LIN {X 0,Y 361.866,Z 148.406,A -85,B 0,C 180,E1 -12924.654,E2 -12924.654} C_VEL
LIN {X 0,Y 361.829,Z 148.411,A -85,B 0,C 180,E1 -12928.369,E2 -12928.369} C_VEL
LIN {X 0,Y 361.892,Z 148.404,A -85,B 0,C 180,E1 -12930.954,E2 -12930.954} C_VEL
LIN {X 0,Y 361.9,Z 148.402,A -85,B 0,C 180,E1 -12934.708,E2 -12934.708} C_VEL
LIN {X 0,Y 361.851,Z 148.408,A -85,B 0,C 180,E1 -12938.344,E2 -12938.344} C_VEL
LIN {X 0,Y 361.91,Z 148.401,A -85,B 0,C 180,E1 -12942.084,E2 -12942.084} C_VEL
LIN {X 0,Y 361.95,Z 148.402,A -85,B 0,C 180,E1 -12945.379,E2 -12945.379} C_VEL
LIN {X 0,Y 361.958,Z 148.397,A -85,B 0,C 180,E1 -12948.804,E2 -12948.804} C_VEL
LIN {X 0,Y 362.066,Z 148.381,A -85,B 0,C 180,E1 -12952.191,E2 -12952.191} C_VEL
LIN {X 0,Y 362.076,Z 148.38,A -85,B 0,C 180,E1 -12954.43,E2 -12954.43} C_VEL
LIN {X 0,Y 362.251,Z 148.359,A -85,B 0,C 180,E1 -12957.776,E2 -12957.776} C_VEL
LIN {X 0,Y 362.252,Z 148.358,A -85,B 0,C 180,E1 -12962.224,E2 -12962.224} C_VEL
LIN {X 0,Y 362.111,Z 148.379,A -85,B 0,C 180,E1 -12966.687,E2 -12966.687} C_VEL
LIN {X 0,Y 361.988,Z 148.391,A -85,B 0,C 180,E1 -12970.063,E2 -12970.063} C_VEL
LIN {X 0,Y 361.987,Z 148.391,A -85,B 0,C 180,E1 -12973.899,E2 -12973.899} C_VEL
LIN {X 0,Y 361.917,Z 148.404,A -85,B 0,C 180,E1 -12976.935,E2 -12976.935} C_VEL
LIN {X 0,Y 361.876,Z 148.409,A -85,B 0,C 180,E1 -12980.462,E2 -12980.462} C_VEL
LIN {X 0,Y 361.883,Z 148.406,A -85,B 0,C 180,E1 -12984.113,E2 -12984.113} C_VEL
LIN {X 0,Y 361.889,Z 148.404,A -85,B 0,C 180,E1 -12987.781,E2 -12987.781} C_VEL
LIN {X 0,Y 361.837,Z 148.41,A -85,B 0,C 180,E1 -12991.286,E2 -12991.286} C_VEL
LIN {X 0,Y 361.845,Z 148.414,A -85,B 0,C 180,E1 -12994.281,E2 -12994.281} C_VEL
LIN {X 0,Y 361.854,Z 148.408,A -85,B 0,C 180,E1 -12997.224,E2 -12997.224} C_VEL
LIN {X 0,Y 361.827,Z 148.413,A -85,B 0,C 180,E1 -13000.756,E2 -13000.756} C_VEL
LIN {X 0,Y 361.81,Z 148.418,A -85,B 0,C 180,E1 -13004.37,E2 -13004.37} C_VEL
LIN {X 0,Y 361.83,Z 148.412,A -85,B 0,C 180,E1 -13007.569,E2 -13007.569} C_VEL
LIN {X 0,Y 361.864,Z 148.406,A -85,B 0,C 180,E1 -13010.975,E2 -13010.975} C_VEL
LIN {X 0,Y 361.87,Z 148.406,A -85,B 0,C 180,E1 -13014.657,E2 -13014.657} C_VEL
LIN {X 0,Y 361.834,Z 148.416,A -85,B 0,C 180,E1 -13018.372,E2 -13018.372} C_VEL
LIN {X 0,Y 361.897,Z 148.42,A -85,B 0,C 180,E1 -13020.133,E2 -13020.133} C_VEL
LIN {X 0,Y 364.194,Z 159.381,A -85,B 0,C 180,E1 -13022.801,E2 -13022.801} C_VEL
LIN {X 0,Y 365.334,Z 165.949,A -85,B 0,C 180,E1 -13024.346,E2 -13024.346} C_VEL
LIN {X 0,Y 364.928,Z 172.793,A -85,B 0,C 180,E1 -13025.844,E2 -13025.844} C_VEL
LIN {X 0,Y 363.854,Z 185.27,A -85,B 0,C 180,E1 -13028.536,E2 -13028.536} C_VEL
LIN {X 0,Y 368.797,Z 220.958,A -85,B 0,C 180,E1 -13029.526,E2 -13029.526} C_VEL
LIN {X 0,Y 367.709,Z 294.28,A -85,B 0,C 180,E1 -13030.971,E2 -13030.971} C_VEL
LIN {X 0,Y 367.075,Z 307.449,A -85,B 0,C 180,E1 -13031.441,E2 -13031.441} C_VEL
LIN {X 0,Y 366.307,Z 320.2,A -85,B 0,C 180,E1 -13032.124,E2 -13032.124} C_VEL
LIN {X 0,Y 365.392,Z 331.51,A -85,B 0,C 180,E1 -13032.944,E2 -13032.944} C_VEL
LIN {X 0,Y 364.323,Z 343.209,A -85,B 0,C 180,E1 -13034.046,E2 -13034.046} C_VEL
LIN {X 0,Y 363.402,Z 353.268,A -85,B 0,C 180,E1 -13035.234,E2 -13035.234} C_VEL
LIN {X 0,Y 362.556,Z 362.347,A -85,B 0,C 180,E1 -13036.55,E2 -13036.55} C_VEL
LIN {X 0,Y 361.857,Z 370.285,A -85,B 0,C 180,E1 -13037.95,E2 -13037.95} C_VEL
LIN {X 0,Y 361.155,Z 378.025,A -85,B 0,C 180,E1 -13039.631,E2 -13039.631} C_VEL
LIN {X 0,Y 360.675,Z 385.162,A -85,B 0,C 180,E1 -13041.598,E2 -13041.598} C_VEL
LIN {X 0,Y 360.482,Z 389.906,A -85,B 0,C 180,E1 -13043.283,E2 -13043.283} C_VEL
LIN {X 0,Y 360.379,Z 393.52,A -85,B 0,C 180,E1 -13044.966,E2 -13044.966} C_VEL
LIN {X 0,Y 360.356,Z 396.112,A -85,B 0,C 180,E1 -13046.647,E2 -13046.647} C_VEL
LIN {X 0,Y 360.396,Z 397.331,A -85,B 0,C 180,E1 -13047.766,E2 -13047.766} C_VEL
LIN {X 0,Y 360.461,Z 398.109,A -85,B 0,C 180,E1 -13048.884,E2 -13048.884} C_VEL
LIN {X 0,Y 360.481,Z 398.478,A -85,B 0,C 180,E1 -13050.001,E2 -13050.001} C_VEL
LIN {X 0,Y 360.456,Z 398.456,A -85,B 0,C 180,E1 -13051.118,E2 -13051.118} C_VEL
LIN {X 0,Y 360.353,Z 398.045,A -85,B 0,C 180,E1 -13052.236,E2 -13052.236} C_VEL
LIN {X 0,Y 360.325,Z 397.214,A -85,B 0,C 180,E1 -13053.355,E2 -13053.355} C_VEL
LIN {X 0,Y 360.36,Z 395.964,A -85,B 0,C 180,E1 -13054.475,E2 -13054.475} C_VEL
LIN {X 0,Y 360.378,Z 393.699,A -85,B 0,C 180,E1 -13055.962,E2 -13055.962} C_VEL
LIN {X 0,Y 360.611,Z 389.673,A -85,B 0,C 180,E1 -13057.842,E2 -13057.842} C_VEL
LIN {X 0,Y 360.997,Z 384.922,A -85,B 0,C 180,E1 -13059.526,E2 -13059.526} C_VEL
LIN {X 0,Y 361.76,Z 377.808,A -85,B 0,C 180,E1 -13061.487,E2 -13061.487} C_VEL
LIN {X 0,Y 362.786,Z 370.109,A -85,B 0,C 180,E1 -13063.158,E2 -13063.158} C_VEL
LIN {X 0,Y 363.776,Z 361.149,A -85,B 0,C 180,E1 -13064.722,E2 -13064.722} C_VEL
LIN {X 0,Y 364.888,Z 351.594,A -85,B 0,C 180,E1 -13066.074,E2 -13066.074} C_VEL
LIN {X 0,Y 366.215,Z 340.759,A -85,B 0,C 180,E1 -13067.306,E2 -13067.306} C_VEL
LIN {X 0,Y 367.436,Z 330.186,A -85,B 0,C 180,E1 -13068.253,E2 -13068.253} C_VEL
LIN {X 0,Y 368.413,Z 319.731,A -85,B 0,C 180,E1 -13068.996,E2 -13068.996} C_VEL
LIN {X 0,Y 369.47,Z 306.271,A -85,B 0,C 180,E1 -13069.698,E2 -13069.698} C_VEL
LIN {X 0,Y 370.177,Z 293.427,A -85,B 0,C 180,E1 -13070.14,E2 -13070.14} C_VEL
LIN {X 0,Y 371.381,Z 220.856,A -85,B 0,C 180,E1 -13071.578,E2 -13071.578} C_VEL
LIN {X 0,Y 366.879,Z 194.148,A -85,B 0,C 180,E1 -13072.44,E2 -13072.44} C_VEL
LIN {X 0,Y 365.076,Z 184.951,A -85,B 0,C 180,E1 -13072.766,E2 -13072.766} C_VEL
LIN {X 0,Y 366.595,Z 171.049,A -85,B 0,C 180,E1 -13075.824,E2 -13075.824} C_VEL
LIN {X 0,Y 365.256,Z 163.227,A -85,B 0,C 180,E1 -13077.736,E2 -13077.736} C_VEL
LIN {X 0,Y 362.77,Z 152.259,A -85,B 0,C 180,E1 -13080.551,E2 -13080.551} C_VEL
LIN {X 0,Y 361.907,Z 148.41,A -85,B 0,C 180,E1 -13081.623,E2 -13081.623} C_VEL
LIN {X 0,Y 361.87,Z 148.411,A -85,B 0,C 180,E1 -13085.637,E2 -13085.637} C_VEL
LIN {X 0,Y 361.866,Z 148.404,A -85,B 0,C 180,E1 -13089.026,E2 -13089.026} C_VEL
LIN {X 0,Y 361.838,Z 148.41,A -85,B 0,C 180,E1 -13092.829,E2 -13092.829} C_VEL
LIN {X 0,Y 361.82,Z 148.416,A -85,B 0,C 180,E1 -13095.947,E2 -13095.947} C_VEL
LIN {X 0,Y 361.814,Z 148.417,A -85,B 0,C 180,E1 -13099.249,E2 -13099.249} C_VEL
LIN {X 0,Y 361.864,Z 148.411,A -85,B 0,C 180,E1 -13102.982,E2 -13102.982} C_VEL
LIN {X 0,Y 361.859,Z 148.412,A -85,B 0,C 180,E1 -13106.631,E2 -13106.631} C_VEL
LIN {X 0,Y 361.857,Z 148.409,A -85,B 0,C 180,E1 -13109.67,E2 -13109.67} C_VEL
LIN {X 0,Y 361.864,Z 148.407,A -85,B 0,C 180,E1 -13113.468,E2 -13113.468} C_VEL
LIN {X 0,Y 361.865,Z 148.409,A -85,B 0,C 180,E1 -13117.143,E2 -13117.143} C_VEL
LIN {X 0,Y 361.855,Z 148.403,A -85,B 0,C 180,E1 -13120.721,E2 -13120.721} C_VEL
LIN {X 0,Y 361.89,Z 148.406,A -85,B 0,C 180,E1 -13124.224,E2 -13124.224} C_VEL
LIN {X 0,Y 361.999,Z 148.386,A -85,B 0,C 180,E1 -13126.528,E2 -13126.528} C_VEL
LIN {X 0,Y 361.994,Z 148.393,A -85,B 0,C 180,E1 -13129.937,E2 -13129.937} C_VEL
LIN {X 0,Y 362.118,Z 148.374,A -85,B 0,C 180,E1 -13133.313,E2 -13133.313} C_VEL
LIN {X 0,Y 362.257,Z 148.351,A -85,B 0,C 180,E1 -13137.776,E2 -13137.776} C_VEL
LIN {X 0,Y 362.173,Z 148.369,A -85,B 0,C 180,E1 -13141.112,E2 -13141.112} C_VEL
LIN {X 0,Y 362.258,Z 148.351,A -85,B 0,C 180,E1 -13142.224,E2 -13142.224} C_VEL
LIN {X 0,Y 362.122,Z 148.374,A -85,B 0,C 180,E1 -13146.687,E2 -13146.687} C_VEL
LIN {X 0,Y 362.001,Z 148.391,A -85,B 0,C 180,E1 -13150.063,E2 -13150.063} C_VEL
LIN {X 0,Y 362,Z 148.382,A -85,B 0,C 180,E1 -13153.899,E2 -13153.899} C_VEL
LIN {X 0,Y 361.929,Z 148.401,A -85,B 0,C 180,E1 -13156.934,E2 -13156.934} C_VEL
LIN {X 0,Y 361.885,Z 148.4,A -85,B 0,C 180,E1 -13160.461,E2 -13160.461} C_VEL
LIN {X 0,Y 361.896,Z 148.397,A -85,B 0,C 180,E1 -13164.113,E2 -13164.113} C_VEL
LIN {X 0,Y 361.863,Z 148.405,A -85,B 0,C 180,E1 -13167.783,E2 -13167.783} C_VEL
LIN {X 0,Y 361.849,Z 148.41,A -85,B 0,C 180,E1 -13171.285,E2 -13171.285} C_VEL
LIN {X 0,Y 361.857,Z 148.409,A -85,B 0,C 180,E1 -13174.28,E2 -13174.28} C_VEL
LIN {X 0,Y 361.865,Z 148.408,A -85,B 0,C 180,E1 -13177.223,E2 -13177.223} C_VEL
LIN {X 0,Y 361.837,Z 148.396,A -85,B 0,C 180,E1 -13180.755,E2 -13180.755} C_VEL
LIN {X 0,Y 361.821,Z 148.416,A -85,B 0,C 180,E1 -13184.368,E2 -13184.368} C_VEL
LIN {X 0,Y 361.836,Z 148.411,A -85,B 0,C 180,E1 -13187.569,E2 -13187.569} C_VEL
LIN {X 0,Y 361.869,Z 148.408,A -85,B 0,C 180,E1 -13190.974,E2 -13190.974} C_VEL
LIN {X 0,Y 361.878,Z 148.408,A -85,B 0,C 180,E1 -13194.655,E2 -13194.655} C_VEL
LIN {X 0,Y 361.842,Z 148.409,A -85,B 0,C 180,E1 -13198.37,E2 -13198.37} C_VEL
LIN {X 0,Y 361.894,Z 148.509,A -85,B 0,C 180,E1 -13200.234,E2 -13200.234} C_VEL
LIN {X 0,Y 363.473,Z 155.472,A -85,B 0,C 180,E1 -13202.171,E2 -13202.171} C_VEL
LIN {X 0,Y 370.386,Z 172.492,A -85,B 0,C 180,E1 -13203.028,E2 -13203.028} C_VEL
LIN {X 0,Y 372.236,Z 181.018,A -85,B 0,C 180,E1 -13203.333,E2 -13203.333} C_VEL
LIN {X 0,Y 370.673,Z 262.367,A -85,B 0,C 180,E1 -13204.935,E2 -13204.935} C_VEL
LIN {X 0,Y 370.018,Z 275.946,A -85,B 0,C 180,E1 -13205.424,E2 -13205.424} C_VEL
LIN {X 0,Y 369.16,Z 288.919,A -85,B 0,C 180,E1 -13206.13,E2 -13206.13} C_VEL
LIN {X 0,Y 368.348,Z 300.168,A -85,B 0,C 180,E1 -13206.974,E2 -13206.974} C_VEL
LIN {X 0,Y 367.174,Z 311.746,A -85,B 0,C 180,E1 -13208.083,E2 -13208.083} C_VEL
LIN {X 0,Y 366.036,Z 321.067,A -85,B 0,C 180,E1 -13209.193,E2 -13209.193} C_VEL
LIN {X 0,Y 364.942,Z 331.045,A -85,B 0,C 180,E1 -13210.672,E2 -13210.672} C_VEL
LIN {X 0,Y 363.824,Z 339.748,A -85,B 0,C 180,E1 -13212.287,E2 -13212.287} C_VEL
LIN {X 0,Y 362.789,Z 347.08,A -85,B 0,C 180,E1 -13213.974,E2 -13213.974} C_VEL
LIN {X 0,Y 361.91,Z 353.714,A -85,B 0,C 180,E1 -13215.931,E2 -13215.931} C_VEL
LIN {X 0,Y 361.358,Z 358.166,A -85,B 0,C 180,E1 -13217.646,E2 -13217.646} C_VEL
LIN {X 0,Y 361.008,Z 360.482,A -85,B 0,C 180,E1 -13218.773,E2 -13218.773} C_VEL
LIN {X 0,Y 360.793,Z 362.366,A -85,B 0,C 180,E1 -13219.902,E2 -13219.902} C_VEL
LIN {X 0,Y 360.655,Z 363.801,A -85,B 0,C 180,E1 -13221.03,E2 -13221.03} C_VEL
LIN {X 0,Y 360.563,Z 365.424,A -85,B 0,C 180,E1 -13223.283,E2 -13223.283} C_VEL
LIN {X 0,Y 360.503,Z 365.665,A -85,B 0,C 180,E1 -13224.405,E2 -13224.405} C_VEL
LIN {X 0,Y 360.478,Z 365.493,A -85,B 0,C 180,E1 -13225.526,E2 -13225.526} C_VEL
LIN {X 0,Y 360.495,Z 363.954,A -85,B 0,C 180,E1 -13227.764,E2 -13227.764} C_VEL
LIN {X 0,Y 360.56,Z 362.608,A -85,B 0,C 180,E1 -13228.882,E2 -13228.882} C_VEL
LIN {X 0,Y 360.722,Z 359.766,A -85,B 0,C 180,E1 -13230.557,E2 -13230.557} C_VEL
LIN {X 0,Y 360.976,Z 355.915,A -85,B 0,C 180,E1 -13232.231,E2 -13232.231} C_VEL
LIN {X 0,Y 361.501,Z 350.939,A -85,B 0,C 180,E1 -13233.901,E2 -13233.901} C_VEL
LIN {X 0,Y 362.073,Z 344.7,A -85,B 0,C 180,E1 -13235.568,E2 -13235.568} C_VEL
LIN {X 0,Y 362.934,Z 336.878,A -85,B 0,C 180,E1 -13237.23,E2 -13237.23} C_VEL
LIN {X 0,Y 363.748,Z 328.918,A -85,B 0,C 180,E1 -13238.611,E2 -13238.611} C_VEL
LIN {X 0,Y 364.686,Z 319.213,A -85,B 0,C 180,E1 -13239.987,E2 -13239.987} C_VEL
LIN {X 0,Y 365.617,Z 308.385,A -85,B 0,C 180,E1 -13241.222,E2 -13241.222} C_VEL
LIN {X 0,Y 366.453,Z 297.773,A -85,B 0,C 180,E1 -13242.178,E2 -13242.178} C_VEL
LIN {X 0,Y 367.184,Z 285.026,A -85,B 0,C 180,E1 -13243.066,E2 -13243.066} C_VEL
LIN {X 0,Y 367.793,Z 272.056,A -85,B 0,C 180,E1 -13243.712,E2 -13243.712} C_VEL
LIN {X 0,Y 368.128,Z 259.143,A -85,B 0,C 180,E1 -13244.122,E2 -13244.122} C_VEL
LIN {X 0,Y 368.76,Z 224.019,A -85,B 0,C 180,E1 -13244.807,E2 -13244.807} C_VEL
LIN {X 0,Y 368.211,Z 218.205,A -85,B 0,C 180,E1 -13244.952,E2 -13244.952} C_VEL
LIN {X 0,Y 363.043,Z 199.491,A -85,B 0,C 180,E1 -13245.605,E2 -13245.605} C_VEL
LIN {X 0,Y 362.507,Z 193.676,A -85,B 0,C 180,E1 -13245.754,E2 -13245.754} C_VEL
LIN {X 0,Y 362.662,Z 178.93,A -85,B 0,C 180,E1 -13246.048,E2 -13246.048} C_VEL
LIN {X 0,Y 359.731,Z 165.344,A -85,B 0,C 180,E1 -13246.495,E2 -13246.495} C_VEL
LIN {X 0,Y 356.068,Z 155.147,A -85,B 0,C 180,E1 -13246.938,E2 -13246.938} C_VEL
LIN {X 0,Y 354.923,Z 149.276,A -85,B 0,C 180,E1 -13248.582,E2 -13248.582} C_VEL
LIN {X 0,Y 354.815,Z 149.288,A -85,B 0,C 180,E1 -13252.106,E2 -13252.106} C_VEL
LIN {X 0,Y 354.897,Z 149.276,A -85,B 0,C 180,E1 -13255.826,E2 -13255.826} C_VEL
LIN {X 0,Y 354.852,Z 149.281,A -85,B 0,C 180,E1 -13259.677,E2 -13259.677} C_VEL
LIN {X 0,Y 354.803,Z 149.288,A -85,B 0,C 180,E1 -13263.701,E2 -13263.701} C_VEL
LIN {X 0,Y 354.795,Z 149.289,A -85,B 0,C 180,E1 -13266.458,E2 -13266.458} C_VEL
LIN {X 0,Y 354.82,Z 149.285,A -85,B 0,C 180,E1 -13269.422,E2 -13269.422} C_VEL
LIN {X 0,Y 354.783,Z 149.288,A -85,B 0,C 180,E1 -13272.866,E2 -13272.866} C_VEL
LIN {X 0,Y 354.761,Z 149.295,A -85,B 0,C 180,E1 -13276.102,E2 -13276.102} C_VEL
LIN {X 0,Y 354.781,Z 149.289,A -85,B 0,C 180,E1 -13279.178,E2 -13279.178} C_VEL
LIN {X 0,Y 354.799,Z 149.287,A -85,B 0,C 180,E1 -13282.402,E2 -13282.402} C_VEL
LIN {X 0,Y 354.804,Z 149.286,A -85,B 0,C 180,E1 -13284.94,E2 -13284.94} C_VEL
LIN {X 0,Y 354.785,Z 149.288,A -85,B 0,C 180,E1 -13288.404,E2 -13288.404} C_VEL
LIN {X 0,Y 354.831,Z 149.288,A -85,B 0,C 180,E1 -13291.617,E2 -13291.617} C_VEL
LIN {X 0,Y 354.865,Z 149.279,A -85,B 0,C 180,E1 -13294.17,E2 -13294.17} C_VEL
LIN {X 0,Y 354.805,Z 149.287,A -85,B 0,C 180,E1 -13297.892,E2 -13297.892} C_VEL
LIN {X 0,Y 354.88,Z 149.278,A -85,B 0,C 180,E1 -13301.907,E2 -13301.907} C_VEL
LIN {X 0,Y 354.932,Z 149.27,A -85,B 0,C 180,E1 -13305.981,E2 -13305.981} C_VEL
LIN {X 0,Y 354.944,Z 149.27,A -85,B 0,C 180,E1 -13309.735,E2 -13309.735} C_VEL
LIN {X 0,Y 355.073,Z 149.258,A -85,B 0,C 180,E1 -13313.179,E2 -13313.179} C_VEL
LIN {X 0,Y 355.213,Z 149.235,A -85,B 0,C 180,E1 -13317.732,E2 -13317.732} C_VEL
LIN {X 0,Y 355.133,Z 149.25,A -85,B 0,C 180,E1 -13321.134,E2 -13321.134} C_VEL
LIN {X 0,Y 355.214,Z 149.235,A -85,B 0,C 180,E1 -13322.268,E2 -13322.268} C_VEL
LIN {X 0,Y 355.076,Z 149.257,A -85,B 0,C 180,E1 -13326.82,E2 -13326.82} C_VEL
LIN {X 0,Y 354.944,Z 149.269,A -85,B 0,C 180,E1 -13330.265,E2 -13330.265} C_VEL
LIN {X 0,Y 354.932,Z 149.27,A -85,B 0,C 180,E1 -13334.019,E2 -13334.019} C_VEL
LIN {X 0,Y 354.879,Z 149.277,A -85,B 0,C 180,E1 -13338.093,E2 -13338.093} C_VEL
LIN {X 0,Y 354.805,Z 149.287,A -85,B 0,C 180,E1 -13342.108,E2 -13342.108} C_VEL
LIN {X 0,Y 354.865,Z 149.278,A -85,B 0,C 180,E1 -13345.83,E2 -13345.83} C_VEL
LIN {X 0,Y 354.845,Z 149.281,A -85,B 0,C 180,E1 -13349.679,E2 -13349.679} C_VEL
LIN {X 0,Y 354.798,Z 149.287,A -85,B 0,C 180,E1 -13353.703,E2 -13353.703} C_VEL
LIN {X 0,Y 354.789,Z 149.293,A -85,B 0,C 180,E1 -13356.461,E2 -13356.461} C_VEL
LIN {X 0,Y 354.816,Z 149.284,A -85,B 0,C 180,E1 -13359.425,E2 -13359.425} C_VEL
LIN {X 0,Y 354.781,Z 149.289,A -85,B 0,C 180,E1 -13362.868,E2 -13362.868} C_VEL
LIN {X 0,Y 354.761,Z 149.297,A -85,B 0,C 180,E1 -13366.105,E2 -13366.105} C_VEL
LIN {X 0,Y 354.782,Z 149.288,A -85,B 0,C 180,E1 -13369.18,E2 -13369.18} C_VEL
LIN {X 0,Y 354.802,Z 149.289,A -85,B 0,C 180,E1 -13372.404,E2 -13372.404} C_VEL
LIN {X 0,Y 354.807,Z 149.285,A -85,B 0,C 180,E1 -13374.942,E2 -13374.942} C_VEL
LIN {X 0,Y 354.79,Z 149.294,A -85,B 0,C 180,E1 -13378.406,E2 -13378.406} C_VEL
LIN {X 0,Y 354.854,Z 149.345,A -85,B 0,C 180,E1 -13379.832,E2 -13379.832} C_VEL
LIN {X 0,Y 357.322,Z 161.045,A -85,B 0,C 180,E1 -13382.742,E2 -13382.742} C_VEL
LIN {X 0,Y 358.436,Z 168.19,A -85,B 0,C 180,E1 -13384.447,E2 -13384.447} C_VEL
LIN {X 0,Y 357.165,Z 182.663,A -85,B 0,C 180,E1 -13387.643,E2 -13387.643} C_VEL
LIN {X 0,Y 356.935,Z 184.932,A -85,B 0,C 180,E1 -13388.139,E2 -13388.139} C_VEL
LIN {X 0,Y 361.814,Z 219.463,A -85,B 0,C 180,E1 -13389.13,E2 -13389.13} C_VEL
LIN {X 0,Y 362.034,Z 226.1,A -85,B 0,C 180,E1 -13389.278,E2 -13389.278} C_VEL
LIN {X 0,Y 360.934,Z 293.87,A -85,B 0,C 180,E1 -13390.637,E2 -13390.637} C_VEL
LIN {X 0,Y 360.284,Z 307.058,A -85,B 0,C 180,E1 -13391.115,E2 -13391.115} C_VEL
LIN {X 0,Y 359.516,Z 319.257,A -85,B 0,C 180,E1 -13391.775,E2 -13391.775} C_VEL
LIN {X 0,Y 358.596,Z 330.743,A -85,B 0,C 180,E1 -13392.611,E2 -13392.611} C_VEL
LIN {X 0,Y 357.472,Z 342.534,A -85,B 0,C 180,E1 -13393.732,E2 -13393.732} C_VEL
LIN {X 0,Y 356.386,Z 353.719,A -85,B 0,C 180,E1 -13395.081,E2 -13395.081} C_VEL
LIN {X 0,Y 355.631,Z 361.782,A -85,B 0,C 180,E1 -13396.283,E2 -13396.283} C_VEL
LIN {X 0,Y 354.866,Z 369.76,A -85,B 0,C 180,E1 -13397.709,E2 -13397.709} C_VEL
LIN {X 0,Y 354.123,Z 377.548,A -85,B 0,C 180,E1 -13399.423,E2 -13399.423} C_VEL
LIN {X 0,Y 353.619,Z 384.715,A -85,B 0,C 180,E1 -13401.429,E2 -13401.429} C_VEL
LIN {X 0,Y 353.392,Z 389.484,A -85,B 0,C 180,E1 -13403.148,E2 -13403.148} C_VEL
LIN {X 0,Y 353.282,Z 393.124,A -85,B 0,C 180,E1 -13404.865,E2 -13404.865} C_VEL
LIN {X 0,Y 353.275,Z 395.74,A -85,B 0,C 180,E1 -13406.58,E2 -13406.58} C_VEL
LIN {X 0,Y 353.297,Z 396.971,A -85,B 0,C 180,E1 -13407.721,E2 -13407.721} C_VEL
LIN {X 0,Y 353.364,Z 397.769,A -85,B 0,C 180,E1 -13408.861,E2 -13408.861} C_VEL
LIN {X 0,Y 353.4,Z 398.149,A -85,B 0,C 180,E1 -13410.001,E2 -13410.001} C_VEL
LIN {X 0,Y 353.357,Z 398.137,A -85,B 0,C 180,E1 -13411.141,E2 -13411.141} C_VEL
LIN {X 0,Y 353.255,Z 397.737,A -85,B 0,C 180,E1 -13412.281,E2 -13412.281} C_VEL
LIN {X 0,Y 353.244,Z 396.927,A -85,B 0,C 180,E1 -13413.423,E2 -13413.423} C_VEL
LIN {X 0,Y 353.27,Z 395.688,A -85,B 0,C 180,E1 -13414.565,E2 -13414.565} C_VEL
LIN {X 0,Y 353.272,Z 393.744,A -85,B 0,C 180,E1 -13415.899,E2 -13415.899} C_VEL
LIN {X 0,Y 353.548,Z 389.443,A -85,B 0,C 180,E1 -13418,E2 -13418} C_VEL
LIN {X 0,Y 353.97,Z 384.717,A -85,B 0,C 180,E1 -13419.717,E2 -13419.717} C_VEL
LIN {X 0,Y 354.775,Z 377.633,A -85,B 0,C 180,E1 -13421.716,E2 -13421.716} C_VEL
LIN {X 0,Y 355.85,Z 369.978,A -85,B 0,C 180,E1 -13423.419,E2 -13423.419} C_VEL
LIN {X 0,Y 356.952,Z 360.632,A -85,B 0,C 180,E1 -13425.081,E2 -13425.081} C_VEL
LIN {X 0,Y 358.213,Z 350.491,A -85,B 0,C 180,E1 -13426.529,E2 -13426.529} C_VEL
LIN {X 0,Y 359.622,Z 339.415,A -85,B 0,C 180,E1 -13427.78,E2 -13427.78} C_VEL
LIN {X 0,Y 360.884,Z 328.579,A -85,B 0,C 180,E1 -13428.744,E2 -13428.744} C_VEL
LIN {X 0,Y 362.059,Z 316.639,A -85,B 0,C 180,E1 -13429.564,E2 -13429.564} C_VEL
LIN {X 0,Y 363.022,Z 303.678,A -85,B 0,C 180,E1 -13430.21,E2 -13430.21} C_VEL
LIN {X 0,Y 363.649,Z 290.822,A -85,B 0,C 180,E1 -13430.617,E2 -13430.617} C_VEL
LIN {X 0,Y 364.924,Z 222.57,A -85,B 0,C 180,E1 -13431.978,E2 -13431.978} C_VEL
LIN {X 0,Y 360.899,Z 197.766,A -85,B 0,C 180,E1 -13432.788,E2 -13432.788} C_VEL
LIN {X 0,Y 358.307,Z 184.595,A -85,B 0,C 180,E1 -13433.27,E2 -13433.27} C_VEL
LIN {X 0,Y 359.724,Z 172.373,A -85,B 0,C 180,E1 -13436.011,E2 -13436.011} C_VEL
LIN {X 0,Y 357.952,Z 162.741,A -85,B 0,C 180,E1 -13438.433,E2 -13438.433} C_VEL
LIN {X 0,Y 354.854,Z 149.29,A -85,B 0,C 180,E1 -13442.02,E2 -13442.02} C_VEL
LIN {X 0,Y 354.824,Z 149.29,A -85,B 0,C 180,E1 -13445.7,E2 -13445.7} C_VEL
LIN {X 0,Y 354.827,Z 149.281,A -85,B 0,C 180,E1 -13449.424,E2 -13449.424} C_VEL
LIN {X 0,Y 354.79,Z 149.288,A -85,B 0,C 180,E1 -13452.867,E2 -13452.867} C_VEL
LIN {X 0,Y 354.768,Z 149.293,A -85,B 0,C 180,E1 -13456.104,E2 -13456.104} C_VEL
LIN {X 0,Y 354.767,Z 149.295,A -85,B 0,C 180,E1 -13459.176,E2 -13459.176} C_VEL
LIN {X 0,Y 354.801,Z 149.289,A -85,B 0,C 180,E1 -13462.405,E2 -13462.405} C_VEL
LIN {X 0,Y 354.81,Z 149.29,A -85,B 0,C 180,E1 -13464.941,E2 -13464.941} C_VEL
LIN {X 0,Y 354.795,Z 149.29,A -85,B 0,C 180,E1 -13468.405,E2 -13468.405} C_VEL
LIN {X 0,Y 354.801,Z 149.287,A -85,B 0,C 180,E1 -13471.615,E2 -13471.615} C_VEL
LIN {X 0,Y 354.836,Z 149.283,A -85,B 0,C 180,E1 -13475.657,E2 -13475.657} C_VEL
LIN {X 0,Y 354.822,Z 149.281,A -85,B 0,C 180,E1 -13479.113,E2 -13479.113} C_VEL
LIN {X 0,Y 354.852,Z 149.284,A -85,B 0,C 180,E1 -13482.718,E2 -13482.718} C_VEL
LIN {X 0,Y 354.94,Z 149.263,A -85,B 0,C 180,E1 -13486.255,E2 -13486.255} C_VEL
LIN {X 0,Y 354.95,Z 149.27,A -85,B 0,C 180,E1 -13489.735,E2 -13489.735} C_VEL
LIN {X 0,Y 355.085,Z 149.25,A -85,B 0,C 180,E1 -13493.18,E2 -13493.18} C_VEL
LIN {X 0,Y 355.218,Z 149.227,A -85,B 0,C 180,E1 -13497.732,E2 -13497.732} C_VEL
LIN {X 0,Y 355.145,Z 149.244,A -85,B 0,C 180,E1 -13501.134,E2 -13501.134} C_VEL
LIN {X 0,Y 355.22,Z 149.227,A -85,B 0,C 180,E1 -13502.268,E2 -13502.268} C_VEL
LIN {X 0,Y 355.088,Z 149.251,A -85,B 0,C 180,E1 -13506.82,E2 -13506.82} C_VEL
LIN {X 0,Y 354.957,Z 149.267,A -85,B 0,C 180,E1 -13510.265,E2 -13510.265} C_VEL
LIN {X 0,Y 354.945,Z 149.26,A -85,B 0,C 180,E1 -13514.019,E2 -13514.019} C_VEL
LIN {X 0,Y 354.892,Z 149.274,A -85,B 0,C 180,E1 -13518.092,E2 -13518.092} C_VEL
LIN {X 0,Y 354.817,Z 149.285,A -85,B 0,C 180,E1 -13522.107,E2 -13522.107} C_VEL
LIN {X 0,Y 354.828,Z 149.284,A -85,B 0,C 180,E1 -13525.833,E2 -13525.833} C_VEL
LIN {X 0,Y 354.81,Z 149.285,A -85,B 0,C 180,E1 -13529.683,E2 -13529.683} C_VEL
LIN {X 0,Y 354.817,Z 149.284,A -85,B 0,C 180,E1 -13533.684,E2 -13533.684} C_VEL
LIN {X 0,Y 354.8,Z 149.286,A -85,B 0,C 180,E1 -13536.46,E2 -13536.46} C_VEL
LIN {X 0,Y 354.827,Z 149.28,A -85,B 0,C 180,E1 -13539.424,E2 -13539.424} C_VEL
LIN {X 0,Y 354.791,Z 149.287,A -85,B 0,C 180,E1 -13542.867,E2 -13542.867} C_VEL
LIN {X 0,Y 354.77,Z 149.294,A -85,B 0,C 180,E1 -13546.103,E2 -13546.103} C_VEL
LIN {X 0,Y 354.787,Z 149.29,A -85,B 0,C 180,E1 -13549.178,E2 -13549.178} C_VEL
LIN {X 0,Y 354.81,Z 149.289,A -85,B 0,C 180,E1 -13552.403,E2 -13552.403} C_VEL
LIN {X 0,Y 354.816,Z 149.288,A -85,B 0,C 180,E1 -13554.941,E2 -13554.941} C_VEL
LIN {X 0,Y 354.797,Z 149.287,A -85,B 0,C 180,E1 -13558.405,E2 -13558.405} C_VEL
LIN {X 0,Y 354.872,Z 149.464,A -85,B 0,C 180,E1 -13559.831,E2 -13559.831} C_VEL
LIN {X 0,Y 356.321,Z 155.683,A -85,B 0,C 180,E1 -13561.634,E2 -13561.634} C_VEL
LIN {X 0,Y 364.068,Z 174.56,A -85,B 0,C 180,E1 -13562.622,E2 -13562.622} C_VEL
LIN {X 0,Y 365.745,Z 181.421,A -85,B 0,C 180,E1 -13562.888,E2 -13562.888} C_VEL
LIN {X 0,Y 364.092,Z 263.039,A -85,B 0,C 180,E1 -13564.526,E2 -13564.526} C_VEL
LIN {X 0,Y 363.43,Z 276.633,A -85,B 0,C 180,E1 -13565.031,E2 -13565.031} C_VEL
LIN {X 0,Y 362.618,Z 288.293,A -85,B 0,C 180,E1 -13565.671,E2 -13565.671} C_VEL
LIN {X 0,Y 361.77,Z 299.814,A -85,B 0,C 180,E1 -13566.531,E2 -13566.531} C_VEL
LIN {X 0,Y 360.546,Z 311.518,A -85,B 0,C 180,E1 -13567.659,E2 -13567.659} C_VEL
LIN {X 0,Y 359.359,Z 320.934,A -85,B 0,C 180,E1 -13568.788,E2 -13568.788} C_VEL
LIN {X 0,Y 358.199,Z 330.74,A -85,B 0,C 180,E1 -13570.247,E2 -13570.247} C_VEL
LIN {X 0,Y 357.006,Z 339.784,A -85,B 0,C 180,E1 -13571.937,E2 -13571.937} C_VEL
LIN {X 0,Y 355.913,Z 347.167,A -85,B 0,C 180,E1 -13573.656,E2 -13573.656} C_VEL
LIN {X 0,Y 355.163,Z 352.164,A -85,B 0,C 180,E1 -13575.092,E2 -13575.092} C_VEL
LIN {X 0,Y 354.502,Z 356.994,A -85,B 0,C 180,E1 -13576.821,E2 -13576.821} C_VEL
LIN {X 0,Y 354.008,Z 360.693,A -85,B 0,C 180,E1 -13578.548,E2 -13578.548} C_VEL
LIN {X 0,Y 353.739,Z 362.596,A -85,B 0,C 180,E1 -13579.699,E2 -13579.699} C_VEL
LIN {X 0,Y 353.587,Z 364.065,A -85,B 0,C 180,E1 -13580.85,E2 -13580.85} C_VEL
LIN {X 0,Y 353.49,Z 365.722,A -85,B 0,C 180,E1 -13583.148,E2 -13583.148} C_VEL
LIN {X 0,Y 353.427,Z 365.98,A -85,B 0,C 180,E1 -13584.293,E2 -13584.293} C_VEL
LIN {X 0,Y 353.409,Z 365.841,A -85,B 0,C 180,E1 -13585.437,E2 -13585.437} C_VEL
LIN {X 0,Y 353.397,Z 364.338,A -85,B 0,C 180,E1 -13587.72,E2 -13587.72} C_VEL
LIN {X 0,Y 353.493,Z 363.007,A -85,B 0,C 180,E1 -13588.86,E2 -13588.86} C_VEL
LIN {X 0,Y 353.639,Z 360.203,A -85,B 0,C 180,E1 -13590.568,E2 -13590.568} C_VEL
LIN {X 0,Y 353.908,Z 356.39,A -85,B 0,C 180,E1 -13592.275,E2 -13592.275} C_VEL
LIN {X 0,Y 354.432,Z 351.455,A -85,B 0,C 180,E1 -13593.978,E2 -13593.978} C_VEL
LIN {X 0,Y 355.05,Z 345.266,A -85,B 0,C 180,E1 -13595.679,E2 -13595.679} C_VEL
LIN {X 0,Y 355.937,Z 337.515,A -85,B 0,C 180,E1 -13597.373,E2 -13597.373} C_VEL
LIN {X 0,Y 356.772,Z 329.617,A -85,B 0,C 180,E1 -13598.78,E2 -13598.78} C_VEL
LIN {X 0,Y 357.819,Z 318.987,A -85,B 0,C 180,E1 -13600.316,E2 -13600.316} C_VEL
LIN {X 0,Y 358.77,Z 308.181,A -85,B 0,C 180,E1 -13601.553,E2 -13601.553} C_VEL
LIN {X 0,Y 359.705,Z 297.088,A -85,B 0,C 180,E1 -13602.553,E2 -13602.553} C_VEL
LIN {X 0,Y 360.38,Z 285.183,A -85,B 0,C 180,E1 -13603.389,E2 -13603.389} C_VEL
LIN {X 0,Y 360.993,Z 272.982,A -85,B 0,C 180,E1 -13604.012,E2 -13604.012} C_VEL
LIN {X 0,Y 361.347,Z 260.511,A -85,B 0,C 180,E1 -13604.429,E2 -13604.429} C_VEL
LIN {X 0,Y 362.507,Z 193.676,A -85,B 0,C 180,E1 -13605.754,E2 -13605.754} C_VEL
LIN {X 0,Y 361.897,Z 187.877,A -85,B 0,C 180,E1 -13605.906,E2 -13605.906} C_VEL
LIN {X 0,Y 360.221,Z 182.318,A -85,B 0,C 180,E1 -13606.115,E2 -13606.115} C_VEL
LIN {X 0,Y 352.169,Z 164.496,A -85,B 0,C 180,E1 -13606.957,E2 -13606.957} C_VEL
LIN {X 0,Y 348.908,Z 155.398,A -85,B 0,C 180,E1 -13607.385,E2 -13607.385} C_VEL
LIN {X 0,Y 347.874,Z 150.152,A -85,B 0,C 180,E1 -13608.858,E2 -13608.858} C_VEL
LIN {X 0,Y 347.762,Z 150.167,A -85,B 0,C 180,E1 -13612.579,E2 -13612.579} C_VEL
LIN {X 0,Y 347.81,Z 150.157,A -85,B 0,C 180,E1 -13615.107,E2 -13615.107} C_VEL
LIN {X 0,Y 347.809,Z 150.159,A -85,B 0,C 180,E1 -13617.692,E2 -13617.692} C_VEL
LIN {X 0,Y 347.762,Z 150.167,A -85,B 0,C 180,E1 -13620.345,E2 -13620.345} C_VEL
LIN {X 0,Y 347.741,Z 150.168,A -85,B 0,C 180,E1 -13624.462,E2 -13624.462} C_VEL
LIN {X 0,Y 347.77,Z 150.168,A -85,B 0,C 180,E1 -13627.987,E2 -13627.987} C_VEL
LIN {X 0,Y 347.746,Z 150.17,A -85,B 0,C 180,E1 -13631.829,E2 -13631.829} C_VEL
LIN {X 0,Y 347.7,Z 150.171,A -85,B 0,C 180,E1 -13635.025,E2 -13635.025} C_VEL
LIN {X 0,Y 347.744,Z 150.166,A -85,B 0,C 180,E1 -13638.396,E2 -13638.396} C_VEL
LIN {X 0,Y 347.766,Z 150.166,A -85,B 0,C 180,E1 -13642.01,E2 -13642.01} C_VEL
LIN {X 0,Y 347.736,Z 150.171,A -85,B 0,C 180,E1 -13645.535,E2 -13645.535} C_VEL
LIN {X 0,Y 347.755,Z 150.17,A -85,B 0,C 180,E1 -13649.652,E2 -13649.652} C_VEL
LIN {X 0,Y 347.814,Z 150.156,A -85,B 0,C 180,E1 -13652.753,E2 -13652.753} C_VEL
LIN {X 0,Y 347.774,Z 150.162,A -85,B 0,C 180,E1 -13656.161,E2 -13656.161} C_VEL
LIN {X 0,Y 347.789,Z 150.161,A -85,B 0,C 180,E1 -13659.908,E2 -13659.908} C_VEL
LIN {X 0,Y 347.82,Z 150.159,A -85,B 0,C 180,E1 -13663.568,E2 -13663.568} C_VEL
LIN {X 0,Y 347.878,Z 150.153,A -85,B 0,C 180,E1 -13667.16,E2 -13667.16} C_VEL
LIN {X 0,Y 347.924,Z 150.144,A -85,B 0,C 180,E1 -13670.7,E2 -13670.7} C_VEL
LIN {X 0,Y 348.024,Z 150.128,A -85,B 0,C 180,E1 -13674.205,E2 -13674.205} C_VEL
LIN {X 0,Y 348.175,Z 150.112,A -85,B 0,C 180,E1 -13677.686,E2 -13677.686} C_VEL
LIN {X 0,Y 348.104,Z 150.125,A -85,B 0,C 180,E1 -13681.157,E2 -13681.157} C_VEL
LIN {X 0,Y 348.176,Z 150.112,A -85,B 0,C 180,E1 -13682.314,E2 -13682.314} C_VEL
LIN {X 0,Y 348.043,Z 150.134,A -85,B 0,C 180,E1 -13686.959,E2 -13686.959} C_VEL
LIN {X 0,Y 347.884,Z 150.15,A -85,B 0,C 180,E1 -13690.476,E2 -13690.476} C_VEL
LIN {X 0,Y 347.888,Z 150.148,A -85,B 0,C 180,E1 -13694.15,E2 -13694.15} C_VEL
LIN {X 0,Y 347.818,Z 150.158,A -85,B 0,C 180,E1 -13698.259,E2 -13698.259} C_VEL
LIN {X 0,Y 347.757,Z 150.164,A -85,B 0,C 180,E1 -13701.627,E2 -13701.627} C_VEL
LIN {X 0,Y 347.789,Z 150.161,A -85,B 0,C 180,E1 -13705.11,E2 -13705.11} C_VEL
LIN {X 0,Y 347.792,Z 150.16,A -85,B 0,C 180,E1 -13707.695,E2 -13707.695} C_VEL
LIN {X 0,Y 347.755,Z 150.169,A -85,B 0,C 180,E1 -13710.347,E2 -13710.347} C_VEL
LIN {X 0,Y 347.736,Z 150.172,A -85,B 0,C 180,E1 -13714.465,E2 -13714.465} C_VEL
LIN {X 0,Y 347.765,Z 150.166,A -85,B 0,C 180,E1 -13717.99,E2 -13717.99} C_VEL
LIN {X 0,Y 347.743,Z 150.167,A -85,B 0,C 180,E1 -13721.831,E2 -13721.831} C_VEL
LIN {X 0,Y 347.699,Z 150.171,A -85,B 0,C 180,E1 -13725.028,E2 -13725.028} C_VEL
LIN {X 0,Y 347.745,Z 150.168,A -85,B 0,C 180,E1 -13728.398,E2 -13728.398} C_VEL
LIN {X 0,Y 347.769,Z 150.168,A -85,B 0,C 180,E1 -13732.013,E2 -13732.013} C_VEL
LIN {X 0,Y 347.74,Z 150.168,A -85,B 0,C 180,E1 -13735.537,E2 -13735.537} C_VEL
LIN {X 0,Y 347.835,Z 150.341,A -85,B 0,C 180,E1 -13739.536,E2 -13739.536} C_VEL
LIN {X 0,Y 350.329,Z 162.073,A -85,B 0,C 180,E1 -13742.524,E2 -13742.524} C_VEL
LIN {X 0,Y 351.499,Z 169.376,A -85,B 0,C 180,E1 -13744.306,E2 -13744.306} C_VEL
LIN {X 0,Y 350.153,Z 183.935,A -85,B 0,C 180,E1 -13747.584,E2 -13747.584} C_VEL
LIN {X 0,Y 350.079,Z 184.593,A -85,B 0,C 180,E1 -13747.731,E2 -13747.731} C_VEL
LIN {X 0,Y 354.594,Z 216.495,A -85,B 0,C 180,E1 -13748.676,E2 -13748.676} C_VEL
LIN {X 0,Y 355.344,Z 223.186,A -85,B 0,C 180,E1 -13748.857,E2 -13748.857} C_VEL
LIN {X 0,Y 354.194,Z 293.329,A -85,B 0,C 180,E1 -13750.288,E2 -13750.288} C_VEL
LIN {X 0,Y 353.481,Z 306.655,A -85,B 0,C 180,E1 -13750.775,E2 -13750.775} C_VEL
LIN {X 0,Y 352.659,Z 319.446,A -85,B 0,C 180,E1 -13751.483,E2 -13751.483} C_VEL
LIN {X 0,Y 351.631,Z 331.588,A -85,B 0,C 180,E1 -13752.405,E2 -13752.405} C_VEL
LIN {X 0,Y 350.494,Z 343.155,A -85,B 0,C 180,E1 -13753.548,E2 -13753.548} C_VEL
LIN {X 0,Y 349.436,Z 353.583,A -85,B 0,C 180,E1 -13754.845,E2 -13754.845} C_VEL
LIN {X 0,Y 348.49,Z 362.944,A -85,B 0,C 180,E1 -13756.294,E2 -13756.294} C_VEL
LIN {X 0,Y 347.607,Z 372.022,A -85,B 0,C 180,E1 -13758.041,E2 -13758.041} C_VEL
LIN {X 0,Y 346.927,Z 379.33,A -85,B 0,C 180,E1 -13759.791,E2 -13759.791} C_VEL
LIN {X 0,Y 346.544,Z 384.266,A -85,B 0,C 180,E1 -13761.252,E2 -13761.252} C_VEL
LIN {X 0,Y 346.318,Z 389.063,A -85,B 0,C 180,E1 -13763.007,E2 -13763.007} C_VEL
LIN {X 0,Y 346.214,Z 392.193,A -85,B 0,C 180,E1 -13764.47,E2 -13764.47} C_VEL
LIN {X 0,Y 346.195,Z 395.368,A -85,B 0,C 180,E1 -13766.51,E2 -13766.51} C_VEL
LIN {X 0,Y 346.2,Z 396.609,A -85,B 0,C 180,E1 -13767.674,E2 -13767.674} C_VEL
LIN {X 0,Y 346.268,Z 397.429,A -85,B 0,C 180,E1 -13768.838,E2 -13768.838} C_VEL
LIN {X 0,Y 346.32,Z 397.82,A -85,B 0,C 180,E1 -13770.001,E2 -13770.001} C_VEL
LIN {X 0,Y 346.259,Z 397.819,A -85,B 0,C 180,E1 -13771.164,E2 -13771.164} C_VEL
LIN {X 0,Y 346.165,Z 396.64,A -85,B 0,C 180,E1 -13773.493,E2 -13773.493} C_VEL
LIN {X 0,Y 346.165,Z 395.412,A -85,B 0,C 180,E1 -13774.659,E2 -13774.659} C_VEL
LIN {X 0,Y 346.198,Z 393.688,A -85,B 0,C 180,E1 -13775.886,E2 -13775.886} C_VEL
LIN {X 0,Y 346.379,Z 390.516,A -85,B 0,C 180,E1 -13777.579,E2 -13777.579} C_VEL
LIN {X 0,Y 346.769,Z 386.195,A -85,B 0,C 180,E1 -13779.332,E2 -13779.332} C_VEL
LIN {X 0,Y 347.48,Z 379.684,A -85,B 0,C 180,E1 -13781.374,E2 -13781.374} C_VEL
LIN {X 0,Y 348.518,Z 372.564,A -85,B 0,C 180,E1 -13783.113,E2 -13783.113} C_VEL
LIN {X 0,Y 349.655,Z 363.708,A -85,B 0,C 180,E1 -13784.85,E2 -13784.85} C_VEL
LIN {X 0,Y 350.967,Z 353.662,A -85,B 0,C 180,E1 -13786.431,E2 -13786.431} C_VEL
LIN {X 0,Y 352.369,Z 343.407,A -85,B 0,C 180,E1 -13787.709,E2 -13787.709} C_VEL
LIN {X 0,Y 353.834,Z 332.053,A -85,B 0,C 180,E1 -13788.831,E2 -13788.831} C_VEL
LIN {X 0,Y 354.935,Z 321.261,A -85,B 0,C 180,E1 -13789.671,E2 -13789.671} C_VEL
LIN {X 0,Y 356.004,Z 309.513,A -85,B 0,C 180,E1 -13790.362,E2 -13790.362} C_VEL
LIN {X 0,Y 356.875,Z 296.197,A -85,B 0,C 180,E1 -13790.896,E2 -13790.896} C_VEL
LIN {X 0,Y 357.377,Z 277.279,A -85,B 0,C 180,E1 -13791.332,E2 -13791.332} C_VEL
LIN {X 0,Y 358.356,Z 222.711,A -85,B 0,C 180,E1 -13792.435,E2 -13792.435} C_VEL
LIN {X 0,Y 354.612,Z 199.793,A -85,B 0,C 180,E1 -13793.206,E2 -13793.206} C_VEL
LIN {X 0,Y 351.57,Z 184.153,A -85,B 0,C 180,E1 -13793.813,E2 -13793.813} C_VEL
LIN {X 0,Y 352.789,Z 173.305,A -85,B 0,C 180,E1 -13796.304,E2 -13796.304} C_VEL
LIN {X 0,Y 350.696,Z 162.594,A -85,B 0,C 180,E1 -13799.077,E2 -13799.077} C_VEL
LIN {X 0,Y 347.775,Z 150.169,A -85,B 0,C 180,E1 -13802.53,E2 -13802.53} C_VEL
LIN {X 0,Y 347.772,Z 150.164,A -85,B 0,C 180,E1 -13806.065,E2 -13806.065} C_VEL
LIN {X 0,Y 347.754,Z 150.163,A -85,B 0,C 180,E1 -13808.793,E2 -13808.793} C_VEL
LIN {X 0,Y 347.752,Z 150.167,A -85,B 0,C 180,E1 -13811.831,E2 -13811.831} C_VEL
LIN {X 0,Y 347.707,Z 150.174,A -85,B 0,C 180,E1 -13815.027,E2 -13815.027} C_VEL
LIN {X 0,Y 347.743,Z 150.168,A -85,B 0,C 180,E1 -13818.399,E2 -13818.399} C_VEL
LIN {X 0,Y 347.757,Z 150.168,A -85,B 0,C 180,E1 -13822.679,E2 -13822.679} C_VEL
LIN {X 0,Y 347.75,Z 150.167,A -85,B 0,C 180,E1 -13825.957,E2 -13825.957} C_VEL
LIN {X 0,Y 347.74,Z 150.168,A -85,B 0,C 180,E1 -13829.651,E2 -13829.651} C_VEL
LIN {X 0,Y 347.749,Z 150.165,A -85,B 0,C 180,E1 -13833.601,E2 -13833.601} C_VEL
LIN {X 0,Y 347.764,Z 150.165,A -85,B 0,C 180,E1 -13836.16,E2 -13836.16} C_VEL
LIN {X 0,Y 347.772,Z 150.158,A -85,B 0,C 180,E1 -13839.907,E2 -13839.907} C_VEL
LIN {X 0,Y 347.795,Z 150.16,A -85,B 0,C 180,E1 -13843.567,E2 -13843.567} C_VEL
LIN {X 0,Y 347.884,Z 150.147,A -85,B 0,C 180,E1 -13847.16,E2 -13847.16} C_VEL
LIN {X 0,Y 347.934,Z 150.135,A -85,B 0,C 180,E1 -13850.701,E2 -13850.701} C_VEL
LIN {X 0,Y 348.035,Z 150.135,A -85,B 0,C 180,E1 -13854.205,E2 -13854.205} C_VEL
LIN {X 0,Y 348.156,Z 150.106,A -85,B 0,C 180,E1 -13857.686,E2 -13857.686} C_VEL
LIN {X 0,Y 348.116,Z 150.12,A -85,B 0,C 180,E1 -13861.157,E2 -13861.157} C_VEL
LIN {X 0,Y 348.182,Z 150.103,A -85,B 0,C 180,E1 -13862.314,E2 -13862.314} C_VEL
LIN {X 0,Y 348.055,Z 150.127,A -85,B 0,C 180,E1 -13866.959,E2 -13866.959} C_VEL
LIN {X 0,Y 347.897,Z 150.146,A -85,B 0,C 180,E1 -13870.476,E2 -13870.476} C_VEL
LIN {X 0,Y 347.901,Z 150.137,A -85,B 0,C 180,E1 -13874.15,E2 -13874.15} C_VEL
LIN {X 0,Y 347.831,Z 150.153,A -85,B 0,C 180,E1 -13878.259,E2 -13878.259} C_VEL
LIN {X 0,Y 347.769,Z 150.165,A -85,B 0,C 180,E1 -13881.626,E2 -13881.626} C_VEL
LIN {X 0,Y 347.777,Z 150.16,A -85,B 0,C 180,E1 -13885.111,E2 -13885.111} C_VEL
LIN {X 0,Y 347.748,Z 150.164,A -85,B 0,C 180,E1 -13887.7,E2 -13887.7} C_VEL
LIN {X 0,Y 347.747,Z 150.166,A -85,B 0,C 180,E1 -13890.348,E2 -13890.348} C_VEL
LIN {X 0,Y 347.751,Z 150.165,A -85,B 0,C 180,E1 -13894.044,E2 -13894.044} C_VEL
LIN {X 0,Y 347.764,Z 150.164,A -85,B 0,C 180,E1 -13897.321,E2 -13897.321} C_VEL
LIN {X 0,Y 347.735,Z 150.155,A -85,B 0,C 180,E1 -13900.297,E2 -13900.297} C_VEL
LIN {X 0,Y 347.726,Z 150.169,A -85,B 0,C 180,E1 -13903.408,E2 -13903.408} C_VEL
LIN {X 0,Y 347.728,Z 150.171,A -85,B 0,C 180,E1 -13906.686,E2 -13906.686} C_VEL
LIN {X 0,Y 347.75,Z 150.169,A -85,B 0,C 180,E1 -13910.173,E2 -13910.173} C_VEL
LIN {X 0,Y 347.764,Z 150.165,A -85,B 0,C 180,E1 -13912.679,E2 -13912.679} C_VEL
LIN {X 0,Y 347.752,Z 150.168,A -85,B 0,C 180,E1 -13915.956,E2 -13915.956} C_VEL
LIN {X 0,Y 347.81,Z 150.266,A -85,B 0,C 180,E1 -13919.363,E2 -13919.363} C_VEL
LIN {X 0,Y 349.18,Z 156.084,A -85,B 0,C 180,E1 -13921.077,E2 -13921.077} C_VEL
LIN {X 0,Y 357.717,Z 176.464,A -85,B 0,C 180,E1 -13922.195,E2 -13922.195} C_VEL
LIN {X 0,Y 359.278,Z 182.53,A -85,B 0,C 180,E1 -13922.443,E2 -13922.443} C_VEL
LIN {X 0,Y 357.54,Z 263.724,A -85,B 0,C 180,E1 -13924.103,E2 -13924.103} C_VEL
LIN {X 0,Y 356.875,Z 276.748,A -85,B 0,C 180,E1 -13924.595,E2 -13924.595} C_VEL
LIN {X 0,Y 355.956,Z 289.571,A -85,B 0,C 180,E1 -13925.317,E2 -13925.317} C_VEL
LIN {X 0,Y 355.051,Z 301.063,A -85,B 0,C 180,E1 -13926.214,E2 -13926.214} C_VEL
LIN {X 0,Y 353.77,Z 312.594,A -85,B 0,C 180,E1 -13927.361,E2 -13927.361} C_VEL
LIN {X 0,Y 352.539,Z 321.88,A -85,B 0,C 180,E1 -13928.511,E2 -13928.511} C_VEL
LIN {X 0,Y 351.471,Z 330.507,A -85,B 0,C 180,E1 -13929.822,E2 -13929.822} C_VEL
LIN {X 0,Y 350.456,Z 338.429,A -85,B 0,C 180,E1 -13931.284,E2 -13931.284} C_VEL
LIN {X 0,Y 349.213,Z 346.139,A -85,B 0,C 180,E1 -13933.032,E2 -13933.032} C_VEL
LIN {X 0,Y 348.244,Z 352.297,A -85,B 0,C 180,E1 -13934.789,E2 -13934.789} C_VEL
LIN {X 0,Y 347.528,Z 357.167,A -85,B 0,C 180,E1 -13936.551,E2 -13936.551} C_VEL
LIN {X 0,Y 347.01,Z 360.905,A -85,B 0,C 180,E1 -13938.314,E2 -13938.314} C_VEL
LIN {X 0,Y 346.693,Z 362.827,A -85,B 0,C 180,E1 -13939.487,E2 -13939.487} C_VEL
LIN {X 0,Y 346.533,Z 364.325,A -85,B 0,C 180,E1 -13940.662,E2 -13940.662} C_VEL
LIN {X 0,Y 346.398,Z 366.022,A -85,B 0,C 180,E1 -13943.007,E2 -13943.007} C_VEL
LIN {X 0,Y 346.347,Z 366.296,A -85,B 0,C 180,E1 -13944.176,E2 -13944.176} C_VEL
LIN {X 0,Y 346.32,Z 366.184,A -85,B 0,C 180,E1 -13945.343,E2 -13945.343} C_VEL
LIN {X 0,Y 346.299,Z 364.721,A -85,B 0,C 180,E1 -13947.673,E2 -13947.673} C_VEL
LIN {X 0,Y 346.409,Z 363.407,A -85,B 0,C 180,E1 -13948.836,E2 -13948.836} C_VEL
LIN {X 0,Y 346.559,Z 360.638,A -85,B 0,C 180,E1 -13950.58,E2 -13950.58} C_VEL
LIN {X 0,Y 346.843,Z 356.862,A -85,B 0,C 180,E1 -13952.321,E2 -13952.321} C_VEL
LIN {X 0,Y 347.368,Z 351.969,A -85,B 0,C 180,E1 -13954.06,E2 -13954.06} C_VEL
LIN {X 0,Y 348.03,Z 345.823,A -85,B 0,C 180,E1 -13955.794,E2 -13955.794} C_VEL
LIN {X 0,Y 348.944,Z 338.15,A -85,B 0,C 180,E1 -13957.521,E2 -13957.521} C_VEL
LIN {X 0,Y 349.797,Z 330.315,A -85,B 0,C 180,E1 -13958.957,E2 -13958.957} C_VEL
LIN {X 0,Y 350.772,Z 320.762,A -85,B 0,C 180,E1 -13960.387,E2 -13960.387} C_VEL
LIN {X 0,Y 351.801,Z 310.275,A -85,B 0,C 180,E1 -13961.654,E2 -13961.654} C_VEL
LIN {X 0,Y 352.706,Z 299.866,A -85,B 0,C 180,E1 -13962.66,E2 -13962.66} C_VEL
LIN {X 0,Y 353.502,Z 287.565,A -85,B 0,C 180,E1 -13963.581,E2 -13963.581} C_VEL
LIN {X 0,Y 354.122,Z 274.611,A -85,B 0,C 180,E1 -13964.289,E2 -13964.289} C_VEL
LIN {X 0,Y 354.581,Z 261.85,A -85,B 0,C 180,E1 -13964.747,E2 -13964.747} C_VEL
LIN {X 0,Y 356.062,Z 180.74,A -85,B 0,C 180,E1 -13966.384,E2 -13966.384} C_VEL
LIN {X 0,Y 353.393,Z 167.979,A -85,B 0,C 180,E1 -13966.81,E2 -13966.81} C_VEL
LIN {X 0,Y 352.169,Z 164.496,A -85,B 0,C 180,E1 -13966.957,E2 -13966.957} C_VEL
LIN {X 0,Y 350.257,Z 161.14,A -85,B 0,C 180,E1 -13967.17,E2 -13967.17} C_VEL
LIN {X 0,Y 347.706,Z 158.445,A -85,B 0,C 180,E1 -13967.469,E2 -13967.469} C_VEL
LIN {X 0,Y 344.201,Z 155.52,A -85,B 0,C 180,E1 -13967.989,E2 -13967.989} C_VEL
LIN {X 0,Y 341.524,Z 152.865,A -85,B 0,C 180,E1 -13968.654,E2 -13968.654} C_VEL
LIN {X 0,Y 340.9,Z 151.517,A -85,B 0,C 180,E1 -13969.037,E2 -13969.037} C_VEL
LIN {X 0,Y 340.803,Z 151.033,A -85,B 0,C 180,E1 -13969.264,E2 -13969.264} C_VEL
LIN {X 0,Y 340.72,Z 151.041,A -85,B 0,C 180,E1 -13973.072,E2 -13973.072} C_VEL
LIN {X 0,Y 340.771,Z 151.035,A -85,B 0,C 180,E1 -13975.663,E2 -13975.663} C_VEL
LIN {X 0,Y 340.74,Z 151.043,A -85,B 0,C 180,E1 -13978.318,E2 -13978.318} C_VEL
LIN {X 0,Y 340.701,Z 151.042,A -85,B 0,C 180,E1 -13981.043,E2 -13981.043} C_VEL
LIN {X 0,Y 340.715,Z 151.041,A -85,B 0,C 180,E1 -13985.277,E2 -13985.277} C_VEL
LIN {X 0,Y 340.706,Z 151.044,A -85,B 0,C 180,E1 -13988.385,E2 -13988.385} C_VEL
LIN {X 0,Y 340.694,Z 151.049,A -85,B 0,C 180,E1 -13992.044,E2 -13992.044} C_VEL
LIN {X 0,Y 340.646,Z 151.052,A -85,B 0,C 180,E1 -13996.226,E2 -13996.226} C_VEL
LIN {X 0,Y 340.682,Z 151.05,A -85,B 0,C 180,E1 -13999.752,E2 -13999.752} C_VEL
LIN {X 0,Y 340.697,Z 151.044,A -85,B 0,C 180,E1 -14003.257,E2 -14003.257} C_VEL
LIN {X 0,Y 340.684,Z 151.046,A -85,B 0,C 180,E1 -14006.152,E2 -14006.152} C_VEL
LIN {X 0,Y 340.766,Z 151.035,A -85,B 0,C 180,E1 -14010.331,E2 -14010.331} C_VEL
LIN {X 0,Y 340.771,Z 151.034,A -85,B 0,C 180,E1 -14013.017,E2 -14013.017} C_VEL
LIN {X 0,Y 340.743,Z 151.042,A -85,B 0,C 180,E1 -14015.637,E2 -14015.637} C_VEL
LIN {X 0,Y 340.72,Z 151.046,A -85,B 0,C 180,E1 -14019.472,E2 -14019.472} C_VEL
LIN {X 0,Y 340.782,Z 151.033,A -85,B 0,C 180,E1 -14021.98,E2 -14021.98} C_VEL
LIN {X 0,Y 340.859,Z 151.025,A -85,B 0,C 180,E1 -14025.704,E2 -14025.704} C_VEL
LIN {X 0,Y 340.836,Z 151.03,A -85,B 0,C 180,E1 -14029.305,E2 -14029.305} C_VEL
LIN {X 0,Y 340.988,Z 151.008,A -85,B 0,C 180,E1 -14032.896,E2 -14032.896} C_VEL
LIN {X 0,Y 340.797,Z 151.033,A -85,B 0,C 180,E1 -14035.268,E2 -14035.268} C_VEL
LIN {X 0,Y 341.112,Z 150.992,A -85,B 0,C 180,E1 -14037.638,E2 -14037.638} C_VEL
LIN {X 0,Y 341.075,Z 151,A -85,B 0,C 180,E1 -14041.181,E2 -14041.181} C_VEL
LIN {X 0,Y 341.113,Z 150.992,A -85,B 0,C 180,E1 -14042.361,E2 -14042.361} C_VEL
LIN {X 0,Y 341.004,Z 151.005,A -85,B 0,C 180,E1 -14045.915,E2 -14045.915} C_VEL
LIN {X 0,Y 340.952,Z 151.012,A -85,B 0,C 180,E1 -14048.356,E2 -14048.356} C_VEL
LIN {X 0,Y 340.838,Z 151.025,A -85,B 0,C 180,E1 -14051.9,E2 -14051.9} C_VEL
LIN {X 0,Y 340.806,Z 151.03,A -85,B 0,C 180,E1 -14055.55,E2 -14055.55} C_VEL
LIN {X 0,Y 340.724,Z 151.041,A -85,B 0,C 180,E1 -14059.27,E2 -14059.27} C_VEL
LIN {X 0,Y 340.71,Z 151.044,A -85,B 0,C 180,E1 -14063.074,E2 -14063.074} C_VEL
LIN {X 0,Y 340.749,Z 151.037,A -85,B 0,C 180,E1 -14065.666,E2 -14065.666} C_VEL
LIN {X 0,Y 340.726,Z 151.044,A -85,B 0,C 180,E1 -14068.321,E2 -14068.321} C_VEL
LIN {X 0,Y 340.695,Z 151.045,A -85,B 0,C 180,E1 -14071.045,E2 -14071.045} C_VEL
LIN {X 0,Y 340.709,Z 151.042,A -85,B 0,C 180,E1 -14075.28,E2 -14075.28} C_VEL
LIN {X 0,Y 340.702,Z 151.048,A -85,B 0,C 180,E1 -14078.387,E2 -14078.387} C_VEL
LIN {X 0,Y 340.692,Z 151.048,A -85,B 0,C 180,E1 -14082.047,E2 -14082.047} C_VEL
LIN {X 0,Y 340.645,Z 151.055,A -85,B 0,C 180,E1 -14086.228,E2 -14086.228} C_VEL
LIN {X 0,Y 340.683,Z 151.047,A -85,B 0,C 180,E1 -14089.754,E2 -14089.754} C_VEL
LIN {X 0,Y 340.7,Z 151.044,A -85,B 0,C 180,E1 -14093.26,E2 -14093.26} C_VEL
LIN {X 0,Y 340.69,Z 151.05,A -85,B 0,C 180,E1 -14096.155,E2 -14096.155} C_VEL
LIN {X 0,Y 340.725,Z 151.067,A -85,B 0,C 180,E1 -14099.155,E2 -14099.155} C_VEL
LIN {X 0,Y 343.288,Z 162.893,A -85,B 0,C 180,E1 -14102.243,E2 -14102.243} C_VEL
LIN {X 0,Y 344.543,Z 170.978,A -85,B 0,C 180,E1 -14104.257,E2 -14104.257} C_VEL
LIN {X 0,Y 343.235,Z 184.282,A -85,B 0,C 180,E1 -14107.311,E2 -14107.311} C_VEL
LIN {X 0,Y 347.682,Z 215.585,A -85,B 0,C 180,E1 -14108.263,E2 -14108.263} C_VEL
LIN {X 0,Y 348.65,Z 223.786,A -85,B 0,C 180,E1 -14108.494,E2 -14108.494} C_VEL
LIN {X 0,Y 347.449,Z 292.873,A -85,B 0,C 180,E1 -14109.927,E2 -14109.927} C_VEL
LIN {X 0,Y 346.725,Z 306.247,A -85,B 0,C 180,E1 -14110.424,E2 -14110.424} C_VEL
LIN {X 0,Y 345.911,Z 318.491,A -85,B 0,C 180,E1 -14111.108,E2 -14111.108} C_VEL
LIN {X 0,Y 345.004,Z 329.129,A -85,B 0,C 180,E1 -14111.903,E2 -14111.903} C_VEL
LIN {X 0,Y 343.906,Z 339.848,A -85,B 0,C 180,E1 -14112.918,E2 -14112.918} C_VEL
LIN {X 0,Y 342.731,Z 350.798,A -85,B 0,C 180,E1 -14114.236,E2 -14114.236} C_VEL
LIN {X 0,Y 341.812,Z 360.643,A -85,B 0,C 180,E1 -14115.717,E2 -14115.717} C_VEL
LIN {X 0,Y 340.934,Z 368.701,A -85,B 0,C 180,E1 -14117.198,E2 -14117.198} C_VEL
LIN {X 0,Y 340.064,Z 376.589,A -85,B 0,C 180,E1 -14118.98,E2 -14118.98} C_VEL
LIN {X 0,Y 339.649,Z 381.96,A -85,B 0,C 180,E1 -14120.473,E2 -14120.473} C_VEL
LIN {X 0,Y 339.322,Z 387.19,A -85,B 0,C 180,E1 -14122.264,E2 -14122.264} C_VEL
LIN {X 0,Y 339.169,Z 391.245,A -85,B 0,C 180,E1 -14124.054,E2 -14124.054} C_VEL
LIN {X 0,Y 339.14,Z 393.336,A -85,B 0,C 180,E1 -14125.246,E2 -14125.246} C_VEL
LIN {X 0,Y 339.118,Z 394.995,A -85,B 0,C 180,E1 -14126.437,E2 -14126.437} C_VEL
LIN {X 0,Y 339.107,Z 396.247,A -85,B 0,C 180,E1 -14127.626,E2 -14127.626} C_VEL
LIN {X 0,Y 339.171,Z 397.088,A -85,B 0,C 180,E1 -14128.814,E2 -14128.814} C_VEL
LIN {X 0,Y 339.227,Z 397.491,A -85,B 0,C 180,E1 -14130.001,E2 -14130.001} C_VEL
LIN {X 0,Y 339.161,Z 397.5,A -85,B 0,C 180,E1 -14131.188,E2 -14131.188} C_VEL
LIN {X 0,Y 339.087,Z 396.351,A -85,B 0,C 180,E1 -14133.566,E2 -14133.566} C_VEL
LIN {X 0,Y 339.08,Z 393.743,A -85,B 0,C 180,E1 -14135.8,E2 -14135.8} C_VEL
LIN {X 0,Y 339.332,Z 390.276,A -85,B 0,C 180,E1 -14137.738,E2 -14137.738} C_VEL
LIN {X 0,Y 339.737,Z 385.981,A -85,B 0,C 180,E1 -14139.527,E2 -14139.527} C_VEL
LIN {X 0,Y 340.495,Z 379.498,A -85,B 0,C 180,E1 -14141.611,E2 -14141.611} C_VEL
LIN {X 0,Y 341.589,Z 372.426,A -85,B 0,C 180,E1 -14143.384,E2 -14143.384} C_VEL
LIN {X 0,Y 342.786,Z 363.609,A -85,B 0,C 180,E1 -14145.155,E2 -14145.155} C_VEL
LIN {X 0,Y 344.139,Z 353.618,A -85,B 0,C 180,E1 -14146.767,E2 -14146.767} C_VEL
LIN {X 0,Y 345.596,Z 343.44,A -85,B 0,C 180,E1 -14148.067,E2 -14148.067} C_VEL
LIN {X 0,Y 347.124,Z 332.168,A -85,B 0,C 180,E1 -14149.209,E2 -14149.209} C_VEL
LIN {X 0,Y 348.411,Z 320.496,A -85,B 0,C 180,E1 -14150.132,E2 -14150.132} C_VEL
LIN {X 0,Y 349.544,Z 307.822,A -85,B 0,C 180,E1 -14150.871,E2 -14150.871} C_VEL
LIN {X 0,Y 350.431,Z 294.054,A -85,B 0,C 180,E1 -14151.403,E2 -14151.403} C_VEL
LIN {X 0,Y 351.348,Z 255.848,A -85,B 0,C 180,E1 -14152.219,E2 -14152.219} C_VEL
LIN {X 0,Y 351.898,Z 223.591,A -85,B 0,C 180,E1 -14152.887,E2 -14152.887} C_VEL
LIN {X 0,Y 348.03,Z 200.161,A -85,B 0,C 180,E1 -14153.702,E2 -14153.702} C_VEL
LIN {X 0,Y 344.917,Z 183.861,A -85,B 0,C 180,E1 -14154.338,E2 -14154.338} C_VEL
LIN {X 0,Y 345.908,Z 175.126,A -85,B 0,C 180,E1 -14156.387,E2 -14156.387} C_VEL
LIN {X 0,Y 344.144,Z 165.584,A -85,B 0,C 180,E1 -14158.897,E2 -14158.897} C_VEL
LIN {X 0,Y 341.226,Z 153.07,A -85,B 0,C 180,E1 -14162.387,E2 -14162.387} C_VEL
LIN {X 0,Y 340.711,Z 151.047,A -85,B 0,C 180,E1 -14163.004,E2 -14163.004} C_VEL
LIN {X 0,Y 340.707,Z 151.041,A -85,B 0,C 180,E1 -14166.742,E2 -14166.742} C_VEL
LIN {X 0,Y 340.689,Z 151.046,A -85,B 0,C 180,E1 -14170.247,E2 -14170.247} C_VEL
LIN {X 0,Y 340.654,Z 151.051,A -85,B 0,C 180,E1 -14173.773,E2 -14173.773} C_VEL
LIN {X 0,Y 340.695,Z 151.047,A -85,B 0,C 180,E1 -14177.956,E2 -14177.956} C_VEL
LIN {X 0,Y 340.72,Z 151.044,A -85,B 0,C 180,E1 -14181.771,E2 -14181.771} C_VEL
LIN {X 0,Y 340.724,Z 151.044,A -85,B 0,C 180,E1 -14185.596,E2 -14185.596} C_VEL
LIN {X 0,Y 340.695,Z 151.048,A -85,B 0,C 180,E1 -14188.955,E2 -14188.955} C_VEL
LIN {X 0,Y 340.72,Z 151.044,A -85,B 0,C 180,E1 -14193.013,E2 -14193.013} C_VEL
LIN {X 0,Y 340.741,Z 151.039,A -85,B 0,C 180,E1 -14195.637,E2 -14195.637} C_VEL
LIN {X 0,Y 340.712,Z 151.037,A -85,B 0,C 180,E1 -14199.472,E2 -14199.472} C_VEL
LIN {X 0,Y 340.761,Z 151.033,A -85,B 0,C 180,E1 -14201.979,E2 -14201.979} C_VEL
LIN {X 0,Y 340.81,Z 151.021,A -85,B 0,C 180,E1 -14205.746,E2 -14205.746} C_VEL
LIN {X 0,Y 340.843,Z 151.026,A -85,B 0,C 180,E1 -14209.305,E2 -14209.305} C_VEL
LIN {X 0,Y 341,Z 151.005,A -85,B 0,C 180,E1 -14212.897,E2 -14212.897} C_VEL
LIN {X 0,Y 340.805,Z 151.031,A -85,B 0,C 180,E1 -14215.269,E2 -14215.269} C_VEL
LIN {X 0,Y 341.096,Z 150.985,A -85,B 0,C 180,E1 -14217.638,E2 -14217.638} C_VEL
LIN {X 0,Y 341.087,Z 150.996,A -85,B 0,C 180,E1 -14221.181,E2 -14221.181} C_VEL
LIN {X 0,Y 341.118,Z 150.982,A -85,B 0,C 180,E1 -14222.362,E2 -14222.362} C_VEL
LIN {X 0,Y 340.991,Z 151.007,A -85,B 0,C 180,E1 -14226.471,E2 -14226.471} C_VEL
LIN {X 0,Y 340.883,Z 151.014,A -85,B 0,C 180,E1 -14229.494,E2 -14229.494} C_VEL
LIN {X 0,Y 340.846,Z 151.024,A -85,B 0,C 180,E1 -14233.11,E2 -14233.11} C_VEL
LIN {X 0,Y 340.776,Z 151.035,A -85,B 0,C 180,E1 -14236.782,E2 -14236.782} C_VEL
LIN {X 0,Y 340.736,Z 151.034,A -85,B 0,C 180,E1 -14239.27,E2 -14239.27} C_VEL
LIN {X 0,Y 340.716,Z 151.041,A -85,B 0,C 180,E1 -14243.074,E2 -14243.074} C_VEL
LIN {X 0,Y 340.729,Z 151.041,A -85,B 0,C 180,E1 -14245.668,E2 -14245.668} C_VEL
LIN {X 0,Y 340.734,Z 151.039,A -85,B 0,C 180,E1 -14249.672,E2 -14249.672} C_VEL
LIN {X 0,Y 340.695,Z 151.043,A -85,B 0,C 180,E1 -14253.847,E2 -14253.847} C_VEL
LIN {X 0,Y 340.707,Z 151.041,A -85,B 0,C 180,E1 -14256.742,E2 -14256.742} C_VEL
LIN {X 0,Y 340.69,Z 151.032,A -85,B 0,C 180,E1 -14260.247,E2 -14260.247} C_VEL
LIN {X 0,Y 340.655,Z 151.051,A -85,B 0,C 180,E1 -14263.773,E2 -14263.773} C_VEL
LIN {X 0,Y 340.701,Z 151.045,A -85,B 0,C 180,E1 -14267.955,E2 -14267.955} C_VEL
LIN {X 0,Y 340.736,Z 151.042,A -85,B 0,C 180,E1 -14271.772,E2 -14271.772} C_VEL
LIN {X 0,Y 340.727,Z 151.043,A -85,B 0,C 180,E1 -14275.595,E2 -14275.595} C_VEL
LIN {X 0,Y 340.736,Z 151.073,A -85,B 0,C 180,E1 -14278.872,E2 -14278.872} C_VEL
LIN {X 0,Y 341.996,Z 156.363,A -85,B 0,C 180,E1 -14280.487,E2 -14280.487} C_VEL
LIN {X 0,Y 350.902,Z 177.304,A -85,B 0,C 180,E1 -14281.689,E2 -14281.689} C_VEL
LIN {X 0,Y 352.606,Z 182.568,A -85,B 0,C 180,E1 -14281.939,E2 -14281.939} C_VEL
LIN {X 0,Y 352.748,Z 187.107,A -85,B 0,C 180,E1 -14282.05,E2 -14282.05} C_VEL
LIN {X 0,Y 351.047,Z 263.578,A -85,B 0,C 180,E1 -14283.638,E2 -14283.638} C_VEL
LIN {X 0,Y 350.38,Z 276.637,A -85,B 0,C 180,E1 -14284.134,E2 -14284.134} C_VEL
LIN {X 0,Y 349.451,Z 288.967,A -85,B 0,C 180,E1 -14284.827,E2 -14284.827} C_VEL
LIN {X 0,Y 348.507,Z 300.72,A -85,B 0,C 180,E1 -14285.739,E2 -14285.739} C_VEL
LIN {X 0,Y 347.175,Z 312.374,A -85,B 0,C 180,E1 -14286.907,E2 -14286.907} C_VEL
LIN {X 0,Y 345.873,Z 321.753,A -85,B 0,C 180,E1 -14288.075,E2 -14288.075} C_VEL
LIN {X 0,Y 344.738,Z 330.456,A -85,B 0,C 180,E1 -14289.41,E2 -14289.41} C_VEL
LIN {X 0,Y 343.676,Z 338.44,A -85,B 0,C 180,E1 -14290.901,E2 -14290.901} C_VEL
LIN {X 0,Y 342.345,Z 346.229,A -85,B 0,C 180,E1 -14292.681,E2 -14292.681} C_VEL
LIN {X 0,Y 341.326,Z 352.432,A -85,B 0,C 180,E1 -14294.473,E2 -14294.473} C_VEL
LIN {X 0,Y 340.547,Z 357.46,A -85,B 0,C 180,E1 -14296.32,E2 -14296.32} C_VEL
LIN {X 0,Y 340.015,Z 361.117,A -85,B 0,C 180,E1 -14298.07,E2 -14298.07} C_VEL
LIN {X 0,Y 339.655,Z 363.058,A -85,B 0,C 180,E1 -14299.267,E2 -14299.267} C_VEL
LIN {X 0,Y 339.492,Z 364.58,A -85,B 0,C 180,E1 -14300.466,E2 -14300.466} C_VEL
LIN {X 0,Y 339.357,Z 365.654,A -85,B 0,C 180,E1 -14301.664,E2 -14301.664} C_VEL
LIN {X 0,Y 339.301,Z 366.584,A -85,B 0,C 180,E1 -14303.847,E2 -14303.847} C_VEL
LIN {X 0,Y 339.234,Z 366.522,A -85,B 0,C 180,E1 -14305.245,E2 -14305.245} C_VEL
LIN {X 0,Y 339.187,Z 366.013,A -85,B 0,C 180,E1 -14306.435,E2 -14306.435} C_VEL
LIN {X 0,Y 339.311,Z 363.807,A -85,B 0,C 180,E1 -14308.812,E2 -14308.812} C_VEL
LIN {X 0,Y 339.483,Z 361.072,A -85,B 0,C 180,E1 -14310.592,E2 -14310.592} C_VEL
LIN {X 0,Y 339.779,Z 357.334,A -85,B 0,C 180,E1 -14312.37,E2 -14312.37} C_VEL
LIN {X 0,Y 340.309,Z 352.482,A -85,B 0,C 180,E1 -14314.144,E2 -14314.144} C_VEL
LIN {X 0,Y 341.012,Z 346.378,A -85,B 0,C 180,E1 -14315.913,E2 -14315.913} C_VEL
LIN {X 0,Y 341.955,Z 338.78,A -85,B 0,C 180,E1 -14317.676,E2 -14317.676} C_VEL
LIN {X 0,Y 342.826,Z 331.009,A -85,B 0,C 180,E1 -14319.14,E2 -14319.14} C_VEL
LIN {X 0,Y 343.827,Z 321.531,A -85,B 0,C 180,E1 -14320.6,E2 -14320.6} C_VEL
LIN {X 0,Y 344.89,Z 311.137,A -85,B 0,C 180,E1 -14321.891,E2 -14321.891} C_VEL
LIN {X 0,Y 345.849,Z 300.849,A -85,B 0,C 180,E1 -14322.915,E2 -14322.915} C_VEL
LIN {X 0,Y 346.67,Z 288.828,A -85,B 0,C 180,E1 -14323.854,E2 -14323.854} C_VEL
LIN {X 0,Y 347.301,Z 276.205,A -85,B 0,C 180,E1 -14324.576,E2 -14324.576} C_VEL
LIN {X 0,Y 347.829,Z 263.023,A -85,B 0,C 180,E1 -14325.077,E2 -14325.077} C_VEL
LIN {X 0,Y 349.388,Z 181.518,A -85,B 0,C 180,E1 -14326.76,E2 -14326.76} C_VEL
LIN {X 0,Y 346.949,Z 170.145,A -85,B 0,C 180,E1 -14327.153,E2 -14327.153} C_VEL
LIN {X 0,Y 341.776,Z 155.764,A -85,B 0,C 180,E1 -14327.819,E2 -14327.819} C_VEL
LIN {X 0,Y 340.9,Z 151.517,A -85,B 0,C 180,E1 -14329.037,E2 -14329.037} C_VEL
LIN {X 0,Y 340.444,Z 151.078,A -85,B 0,C 180,E1 -14329.477,E2 -14329.477} C_VEL
LIN {X 0,Y 338.061,Z 151.374,A -85,B 0,C 180,E1 -14330.893,E2 -14330.893} C_VEL
LIN {X 0,Y 334.623,Z 152.002,A -85,B 0,C 180,E1 -14332.875,E2 -14332.875} C_VEL
LIN {X 0,Y 333.732,Z 151.932,A -85,B 0,C 180,E1 -14333.915,E2 -14333.915} C_VEL
LIN {X 0,Y 333.675,Z 151.916,A -85,B 0,C 180,E1 -14334.266,E2 -14334.266} C_VEL
LIN {X 0,Y 333.72,Z 151.915,A -85,B 0,C 180,E1 -14337.809,E2 -14337.809} C_VEL
LIN {X 0,Y 333.695,Z 151.919,A -85,B 0,C 180,E1 -14340.361,E2 -14340.361} C_VEL
LIN {X 0,Y 333.682,Z 151.917,A -85,B 0,C 180,E1 -14344.773,E2 -14344.773} C_VEL
LIN {X 0,Y 333.648,Z 151.923,A -85,B 0,C 180,E1 -14347.65,E2 -14347.65} C_VEL
LIN {X 0,Y 333.642,Z 151.922,A -85,B 0,C 180,E1 -14350.766,E2 -14350.766} C_VEL
LIN {X 0,Y 333.588,Z 151.931,A -85,B 0,C 180,E1 -14354.249,E2 -14354.249} C_VEL
LIN {X 0,Y 333.635,Z 151.926,A -85,B 0,C 180,E1 -14357.617,E2 -14357.617} C_VEL
LIN {X 0,Y 333.646,Z 151.923,A -85,B 0,C 180,E1 -14361.201,E2 -14361.201} C_VEL
LIN {X 0,Y 333.668,Z 151.924,A -85,B 0,C 180,E1 -14363.86,E2 -14363.86} C_VEL
LIN {X 0,Y 333.635,Z 151.926,A -85,B 0,C 180,E1 -14367.412,E2 -14367.412} C_VEL
LIN {X 0,Y 333.699,Z 151.916,A -85,B 0,C 180,E1 -14371.027,E2 -14371.027} C_VEL
LIN {X 0,Y 333.701,Z 151.915,A -85,B 0,C 180,E1 -14374.902,E2 -14374.902} C_VEL
LIN {X 0,Y 333.661,Z 151.92,A -85,B 0,C 180,E1 -14379.018,E2 -14379.018} C_VEL
LIN {X 0,Y 333.731,Z 151.915,A -85,B 0,C 180,E1 -14381.586,E2 -14381.586} C_VEL
LIN {X 0,Y 333.798,Z 151.906,A -85,B 0,C 180,E1 -14385.576,E2 -14385.576} C_VEL
LIN {X 0,Y 333.806,Z 151.906,A -85,B 0,C 180,E1 -14389.077,E2 -14389.077} C_VEL
LIN {X 0,Y 333.944,Z 151.883,A -85,B 0,C 180,E1 -14392.746,E2 -14392.746} C_VEL
LIN {X 0,Y 333.764,Z 151.907,A -85,B 0,C 180,E1 -14395.168,E2 -14395.168} C_VEL
LIN {X 0,Y 334.052,Z 151.872,A -85,B 0,C 180,E1 -14397.588,E2 -14397.588} C_VEL
LIN {X 0,Y 334.046,Z 151.875,A -85,B 0,C 180,E1 -14401.205,E2 -14401.205} C_VEL
LIN {X 0,Y 334.054,Z 151.871,A -85,B 0,C 180,E1 -14402.411,E2 -14402.411} C_VEL
LIN {X 0,Y 333.977,Z 151.88,A -85,B 0,C 180,E1 -14406.04,E2 -14406.04} C_VEL
LIN {X 0,Y 333.809,Z 151.902,A -85,B 0,C 180,E1 -14409.697,E2 -14409.697} C_VEL
LIN {X 0,Y 333.786,Z 151.905,A -85,B 0,C 180,E1 -14413.392,E2 -14413.392} C_VEL
LIN {X 0,Y 333.708,Z 151.916,A -85,B 0,C 180,E1 -14417.148,E2 -14417.148} C_VEL
LIN {X 0,Y 333.661,Z 151.92,A -85,B 0,C 180,E1 -14419.695,E2 -14419.695} C_VEL
LIN {X 0,Y 333.658,Z 151.921,A -85,B 0,C 180,E1 -14423.591,E2 -14423.591} C_VEL
LIN {X 0,Y 333.709,Z 151.917,A -85,B 0,C 180,E1 -14426.248,E2 -14426.248} C_VEL
LIN {X 0,Y 333.699,Z 151.917,A -85,B 0,C 180,E1 -14428.973,E2 -14428.973} C_VEL
LIN {X 0,Y 333.634,Z 151.928,A -85,B 0,C 180,E1 -14432.588,E2 -14432.588} C_VEL
LIN {X 0,Y 333.668,Z 151.923,A -85,B 0,C 180,E1 -14436.14,E2 -14436.14} C_VEL
LIN {X 0,Y 333.639,Z 151.923,A -85,B 0,C 180,E1 -14439.193,E2 -14439.193} C_VEL
LIN {X 0,Y 333.625,Z 151.928,A -85,B 0,C 180,E1 -14442.501,E2 -14442.501} C_VEL
LIN {X 0,Y 333.59,Z 151.932,A -85,B 0,C 180,E1 -14445.956,E2 -14445.956} C_VEL
LIN {X 0,Y 333.642,Z 151.922,A -85,B 0,C 180,E1 -14449.317,E2 -14449.317} C_VEL
LIN {X 0,Y 333.66,Z 151.921,A -85,B 0,C 180,E1 -14453.169,E2 -14453.169} C_VEL
LIN {X 0,Y 333.635,Z 151.926,A -85,B 0,C 180,E1 -14456.793,E2 -14456.793} C_VEL
LIN {X 0,Y 333.678,Z 151.963,A -85,B 0,C 180,E1 -14458.804,E2 -14458.804} C_VEL
LIN {X 0,Y 336.291,Z 163.907,A -85,B 0,C 180,E1 -14462.001,E2 -14462.001} C_VEL
LIN {X 0,Y 337.601,Z 172.046,A -85,B 0,C 180,E1 -14464.078,E2 -14464.078} C_VEL
LIN {X 0,Y 336.395,Z 183.937,A -85,B 0,C 180,E1 -14466.868,E2 -14466.868} C_VEL
LIN {X 0,Y 340.998,Z 215.978,A -85,B 0,C 180,E1 -14467.875,E2 -14467.875} C_VEL
LIN {X 0,Y 341.924,Z 225.473,A -85,B 0,C 180,E1 -14468.138,E2 -14468.138} C_VEL
LIN {X 0,Y 340.655,Z 293.554,A -85,B 0,C 180,E1 -14469.588,E2 -14469.588} C_VEL
LIN {X 0,Y 339.923,Z 306.596,A -85,B 0,C 180,E1 -14470.094,E2 -14470.094} C_VEL
LIN {X 0,Y 339.084,Z 318.666,A -85,B 0,C 180,E1 -14470.791,E2 -14470.791} C_VEL
LIN {X 0,Y 338.074,Z 330.052,A -85,B 0,C 180,E1 -14471.675,E2 -14471.675} C_VEL
LIN {X 0,Y 336.78,Z 341.778,A -85,B 0,C 180,E1 -14472.858,E2 -14472.858} C_VEL
LIN {X 0,Y 335.631,Z 352.332,A -85,B 0,C 180,E1 -14474.205,E2 -14474.205} C_VEL
LIN {X 0,Y 334.672,Z 361.843,A -85,B 0,C 180,E1 -14475.716,E2 -14475.716} C_VEL
LIN {X 0,Y 333.621,Z 370.993,A -85,B 0,C 180,E1 -14477.532,E2 -14477.532} C_VEL
LIN {X 0,Y 332.847,Z 378.367,A -85,B 0,C 180,E1 -14479.354,E2 -14479.354} C_VEL
LIN {X 0,Y 332.444,Z 383.365,A -85,B 0,C 180,E1 -14480.878,E2 -14480.878} C_VEL
LIN {X 0,Y 332.17,Z 388.216,A -85,B 0,C 180,E1 -14482.708,E2 -14482.708} C_VEL
LIN {X 0,Y 332.088,Z 391.126,A -85,B 0,C 180,E1 -14484.079,E2 -14484.079} C_VEL
LIN {X 0,Y 332.042,Z 394.622,A -85,B 0,C 180,E1 -14486.361,E2 -14486.361} C_VEL
LIN {X 0,Y 332.017,Z 395.884,A -85,B 0,C 180,E1 -14487.575,E2 -14487.575} C_VEL
LIN {X 0,Y 332.074,Z 396.744,A -85,B 0,C 180,E1 -14488.788,E2 -14488.788} C_VEL
LIN {X 0,Y 332.134,Z 397.162,A -85,B 0,C 180,E1 -14490.001,E2 -14490.001} C_VEL
LIN {X 0,Y 332.063,Z 397.181,A -85,B 0,C 180,E1 -14491.214,E2 -14491.214} C_VEL
LIN {X 0,Y 332.009,Z 396.06,A -85,B 0,C 180,E1 -14493.642,E2 -14493.642} C_VEL
LIN {X 0,Y 332.001,Z 393.704,A -85,B 0,C 180,E1 -14495.773,E2 -14495.773} C_VEL
LIN {X 0,Y 332.258,Z 390.037,A -85,B 0,C 180,E1 -14497.904,E2 -14497.904} C_VEL
LIN {X 0,Y 332.718,Z 385.767,A -85,B 0,C 180,E1 -14499.73,E2 -14499.73} C_VEL
LIN {X 0,Y 333.518,Z 379.313,A -85,B 0,C 180,E1 -14501.857,E2 -14501.857} C_VEL
LIN {X 0,Y 334.673,Z 372.288,A -85,B 0,C 180,E1 -14503.666,E2 -14503.666} C_VEL
LIN {X 0,Y 335.925,Z 363.512,A -85,B 0,C 180,E1 -14505.472,E2 -14505.472} C_VEL
LIN {X 0,Y 337.331,Z 353.569,A -85,B 0,C 180,E1 -14507.115,E2 -14507.115} C_VEL
LIN {X 0,Y 338.857,Z 343.479,A -85,B 0,C 180,E1 -14508.44,E2 -14508.44} C_VEL
LIN {X 0,Y 340.424,Z 332.289,A -85,B 0,C 180,E1 -14509.602,E2 -14509.602} C_VEL
LIN {X 0,Y 341.645,Z 321.725,A -85,B 0,C 180,E1 -14510.47,E2 -14510.47} C_VEL
LIN {X 0,Y 342.904,Z 309.025,A -85,B 0,C 180,E1 -14511.256,E2 -14511.256} C_VEL
LIN {X 0,Y 343.818,Z 295.958,A -85,B 0,C 180,E1 -14511.803,E2 -14511.803} C_VEL
LIN {X 0,Y 344.337,Z 278.391,A -85,B 0,C 180,E1 -14512.231,E2 -14512.231} C_VEL
LIN {X 0,Y 345.444,Z 224.426,A -85,B 0,C 180,E1 -14513.359,E2 -14513.359} C_VEL
LIN {X 0,Y 341.269,Z 199.43,A -85,B 0,C 180,E1 -14514.259,E2 -14514.259} C_VEL
LIN {X 0,Y 338.171,Z 183.524,A -85,B 0,C 180,E1 -14514.904,E2 -14514.904} C_VEL
LIN {X 0,Y 338.971,Z 177.304,A -85,B 0,C 180,E1 -14516.39,E2 -14516.39} C_VEL
LIN {X 0,Y 338.184,Z 171.639,A -85,B 0,C 180,E1 -14517.879,E2 -14517.879} C_VEL
LIN {X 0,Y 335.62,Z 159.982,A -85,B 0,C 180,E1 -14521.126,E2 -14521.126} C_VEL
LIN {X 0,Y 333.677,Z 151.925,A -85,B 0,C 180,E1 -14523.521,E2 -14523.521} C_VEL
LIN {X 0,Y 333.667,Z 151.917,A -85,B 0,C 180,E1 -14526.832,E2 -14526.832} C_VEL
LIN {X 0,Y 333.648,Z 151.922,A -85,B 0,C 180,E1 -14530.768,E2 -14530.768} C_VEL
LIN {X 0,Y 333.595,Z 151.93,A -85,B 0,C 180,E1 -14534.251,E2 -14534.251} C_VEL
LIN {X 0,Y 333.64,Z 151.927,A -85,B 0,C 180,E1 -14537.618,E2 -14537.618} C_VEL
LIN {X 0,Y 333.636,Z 151.927,A -85,B 0,C 180,E1 -14541.206,E2 -14541.206} C_VEL
LIN {X 0,Y 333.675,Z 151.921,A -85,B 0,C 180,E1 -14543.861,E2 -14543.861} C_VEL
LIN {X 0,Y 333.645,Z 151.926,A -85,B 0,C 180,E1 -14547.413,E2 -14547.413} C_VEL
LIN {X 0,Y 333.654,Z 151.924,A -85,B 0,C 180,E1 -14551.023,E2 -14551.023} C_VEL
LIN {X 0,Y 333.697,Z 151.919,A -85,B 0,C 180,E1 -14555.088,E2 -14555.088} C_VEL
LIN {X 0,Y 333.653,Z 151.918,A -85,B 0,C 180,E1 -14559.017,E2 -14559.017} C_VEL
LIN {X 0,Y 333.713,Z 151.91,A -85,B 0,C 180,E1 -14561.585,E2 -14561.585} C_VEL
LIN {X 0,Y 333.762,Z 151.899,A -85,B 0,C 180,E1 -14565.609,E2 -14565.609} C_VEL
LIN {X 0,Y 333.813,Z 151.902,A -85,B 0,C 180,E1 -14569.077,E2 -14569.077} C_VEL
LIN {X 0,Y 333.956,Z 151.883,A -85,B 0,C 180,E1 -14572.746,E2 -14572.746} C_VEL
LIN {X 0,Y 333.772,Z 151.907,A -85,B 0,C 180,E1 -14575.169,E2 -14575.169} C_VEL
LIN {X 0,Y 334.04,Z 151.864,A -85,B 0,C 180,E1 -14577.588,E2 -14577.588} C_VEL
LIN {X 0,Y 334.058,Z 151.871,A -85,B 0,C 180,E1 -14581.206,E2 -14581.206} C_VEL
LIN {X 0,Y 334.059,Z 151.861,A -85,B 0,C 180,E1 -14582.412,E2 -14582.412} C_VEL
LIN {X 0,Y 333.961,Z 151.882,A -85,B 0,C 180,E1 -14586.462,E2 -14586.462} C_VEL
LIN {X 0,Y 333.822,Z 151.896,A -85,B 0,C 180,E1 -14589.696,E2 -14589.696} C_VEL
LIN {X 0,Y 333.795,Z 151.898,A -85,B 0,C 180,E1 -14593.392,E2 -14593.392} C_VEL
LIN {X 0,Y 333.721,Z 151.917,A -85,B 0,C 180,E1 -14597.148,E2 -14597.148} C_VEL
LIN {X 0,Y 333.673,Z 151.913,A -85,B 0,C 180,E1 -14599.694,E2 -14599.694} C_VEL
LIN {X 0,Y 333.662,Z 151.915,A -85,B 0,C 180,E1 -14603.591,E2 -14603.591} C_VEL
LIN {X 0,Y 333.666,Z 151.92,A -85,B 0,C 180,E1 -14606.252,E2 -14606.252} C_VEL
LIN {X 0,Y 333.667,Z 151.92,A -85,B 0,C 180,E1 -14610.278,E2 -14610.278} C_VEL
LIN {X 0,Y 333.64,Z 151.922,A -85,B 0,C 180,E1 -14613.208,E2 -14613.208} C_VEL
LIN {X 0,Y 333.679,Z 151.917,A -85,B 0,C 180,E1 -14616.139,E2 -14616.139} C_VEL
LIN {X 0,Y 333.65,Z 151.918,A -85,B 0,C 180,E1 -14619.192,E2 -14619.192} C_VEL
LIN {X 0,Y 333.635,Z 151.915,A -85,B 0,C 180,E1 -14622.5,E2 -14622.5} C_VEL
LIN {X 0,Y 333.599,Z 151.929,A -85,B 0,C 180,E1 -14625.955,E2 -14625.955} C_VEL
LIN {X 0,Y 333.65,Z 151.924,A -85,B 0,C 180,E1 -14629.315,E2 -14629.315} C_VEL
LIN {X 0,Y 333.669,Z 151.921,A -85,B 0,C 180,E1 -14633.168,E2 -14633.168} C_VEL
LIN {X 0,Y 333.678,Z 151.921,A -85,B 0,C 180,E1 -14635.341,E2 -14635.341} C_VEL
LIN {X 0,Y 333.702,Z 152.029,A -85,B 0,C 180,E1 -14638.404,E2 -14638.404} C_VEL
LIN {X 0,Y 334.775,Z 156.651,A -85,B 0,C 180,E1 -14639.864,E2 -14639.864} C_VEL
LIN {X 0,Y 344.025,Z 177.887,A -85,B 0,C 180,E1 -14641.15,E2 -14641.15} C_VEL
LIN {X 0,Y 346.311,Z 184.315,A -85,B 0,C 180,E1 -14641.482,E2 -14641.482} C_VEL
LIN {X 0,Y 344.582,Z 263.549,A -85,B 0,C 180,E1 -14643.159,E2 -14643.159} C_VEL
LIN {X 0,Y 343.855,Z 277.222,A -85,B 0,C 180,E1 -14643.687,E2 -14643.687} C_VEL
LIN {X 0,Y 342.872,Z 289.73,A -85,B 0,C 180,E1 -14644.408,E2 -14644.408} C_VEL
LIN {X 0,Y 341.948,Z 300.696,A -85,B 0,C 180,E1 -14645.275,E2 -14645.275} C_VEL
LIN {X 0,Y 340.602,Z 312.157,A -85,B 0,C 180,E1 -14646.434,E2 -14646.434} C_VEL
LIN {X 0,Y 339.22,Z 321.629,A -85,B 0,C 180,E1 -14647.622,E2 -14647.622} C_VEL
LIN {X 0,Y 338.012,Z 330.407,A -85,B 0,C 180,E1 -14648.981,E2 -14648.981} C_VEL
LIN {X 0,Y 336.893,Z 338.454,A -85,B 0,C 180,E1 -14650.501,E2 -14650.501} C_VEL
LIN {X 0,Y 335.496,Z 346.319,A -85,B 0,C 180,E1 -14652.316,E2 -14652.316} C_VEL
LIN {X 0,Y 334.422,Z 352.568,A -85,B 0,C 180,E1 -14654.144,E2 -14654.144} C_VEL
LIN {X 0,Y 333.665,Z 357.273,A -85,B 0,C 180,E1 -14655.874,E2 -14655.874} C_VEL
LIN {X 0,Y 332.994,Z 361.331,A -85,B 0,C 180,E1 -14657.815,E2 -14657.815} C_VEL
LIN {X 0,Y 332.624,Z 363.29,A -85,B 0,C 180,E1 -14659.037,E2 -14659.037} C_VEL
LIN {X 0,Y 332.425,Z 364.83,A -85,B 0,C 180,E1 -14660.262,E2 -14660.262} C_VEL
LIN {X 0,Y 332.282,Z 365.937,A -85,B 0,C 180,E1 -14661.485,E2 -14661.485} C_VEL
LIN {X 0,Y 332.221,Z 366.918,A -85,B 0,C 180,E1 -14663.866,E2 -14663.866} C_VEL
LIN {X 0,Y 332.153,Z 366.855,A -85,B 0,C 180,E1 -14665.144,E2 -14665.144} C_VEL
LIN {X 0,Y 332.11,Z 366.379,A -85,B 0,C 180,E1 -14666.359,E2 -14666.359} C_VEL
LIN {X 0,Y 332.213,Z 364.206,A -85,B 0,C 180,E1 -14668.787,E2 -14668.787} C_VEL
LIN {X 0,Y 332.408,Z 361.505,A -85,B 0,C 180,E1 -14670.605,E2 -14670.605} C_VEL
LIN {X 0,Y 332.718,Z 357.804,A -85,B 0,C 180,E1 -14672.42,E2 -14672.42} C_VEL
LIN {X 0,Y 333.254,Z 352.993,A -85,B 0,C 180,E1 -14674.232,E2 -14674.232} C_VEL
LIN {X 0,Y 333.998,Z 346.931,A -85,B 0,C 180,E1 -14676.038,E2 -14676.038} C_VEL
LIN {X 0,Y 334.97,Z 339.397,A -85,B 0,C 180,E1 -14677.837,E2 -14677.837} C_VEL
LIN {X 0,Y 335.857,Z 331.697,A -85,B 0,C 180,E1 -14679.332,E2 -14679.332} C_VEL
LIN {X 0,Y 336.889,Z 322.297,A -85,B 0,C 180,E1 -14680.82,E2 -14680.82} C_VEL
LIN {X 0,Y 338.032,Z 311.579,A -85,B 0,C 180,E1 -14682.185,E2 -14682.185} C_VEL
LIN {X 0,Y 339.133,Z 300.242,A -85,B 0,C 180,E1 -14683.328,E2 -14683.328} C_VEL
LIN {X 0,Y 339.96,Z 287.848,A -85,B 0,C 180,E1 -14684.286,E2 -14684.286} C_VEL
LIN {X 0,Y 340.662,Z 274.76,A -85,B 0,C 180,E1 -14685.019,E2 -14685.019} C_VEL
LIN {X 0,Y 341.162,Z 261.524,A -85,B 0,C 180,E1 -14685.494,E2 -14685.494} C_VEL
LIN {X 0,Y 342.632,Z 182.015,A -85,B 0,C 180,E1 -14687.161,E2 -14687.161} C_VEL
LIN {X 0,Y 340.557,Z 172.455,A -85,B 0,C 180,E1 -14687.503,E2 -14687.503} C_VEL
LIN {X 0,Y 334.64,Z 156.111,A -85,B 0,C 180,E1 -14688.277,E2 -14688.277} C_VEL
LIN {X 0,Y 333.747,Z 151.913,A -85,B 0,C 180,E1 -14689.559,E2 -14689.559} C_VEL
LIN {X 0,Y 333.668,Z 151.92,A -85,B 0,C 180,E1 -14693.589,E2 -14693.589} C_VEL
LIN {X 0,Y 333.675,Z 151.916,A -85,B 0,C 180,E1 -14694.266,E2 -14694.266} C_VEL
LIN {X 0,Y 333.034,Z 151.999,A -85,B 0,C 180,E1 -14695.273,E2 -14695.273} C_VEL
LIN {X 0,Y 330.157,Z 152.357,A -85,B 0,C 180,E1 -14696.912,E2 -14696.912} C_VEL
LIN {X 0,Y 327.724,Z 152.664,A -85,B 0,C 180,E1 -14698.239,E2 -14698.239} C_VEL
LIN {X 0,Y 326.717,Z 152.785,A -85,B 0,C 180,E1 -14699.268,E2 -14699.268} C_VEL
LIN {X 0,Y 326.656,Z 152.793,A -85,B 0,C 180,E1 -14699.616,E2 -14699.616} C_VEL
LIN {X 0,Y 326.604,Z 152.803,A -85,B 0,C 180,E1 -14704.018,E2 -14704.018} C_VEL
LIN {X 0,Y 326.624,Z 152.796,A -85,B 0,C 180,E1 -14707.237,E2 -14707.237} C_VEL
LIN {X 0,Y 326.573,Z 152.802,A -85,B 0,C 180,E1 -14711.13,E2 -14711.13} C_VEL
LIN {X 0,Y 326.522,Z 152.809,A -85,B 0,C 180,E1 -14714.741,E2 -14714.741} C_VEL
LIN {X 0,Y 326.57,Z 152.806,A -85,B 0,C 180,E1 -14718.153,E2 -14718.153} C_VEL
LIN {X 0,Y 326.616,Z 152.799,A -85,B 0,C 180,E1 -14721.39,E2 -14721.39} C_VEL
LIN {X 0,Y 326.611,Z 152.798,A -85,B 0,C 180,E1 -14724.85,E2 -14724.85} C_VEL
LIN {X 0,Y 326.6,Z 152.802,A -85,B 0,C 180,E1 -14727.454,E2 -14727.454} C_VEL
LIN {X 0,Y 326.651,Z 152.793,A -85,B 0,C 180,E1 -14730.34,E2 -14730.34} C_VEL
LIN {X 0,Y 326.661,Z 152.792,A -85,B 0,C 180,E1 -14733.14,E2 -14733.14} C_VEL
LIN {X 0,Y 326.636,Z 152.797,A -85,B 0,C 180,E1 -14735.87,E2 -14735.87} C_VEL
LIN {X 0,Y 326.613,Z 152.799,A -85,B 0,C 180,E1 -14739.862,E2 -14739.862} C_VEL
LIN {X 0,Y 326.697,Z 152.787,A -85,B 0,C 180,E1 -14743.76,E2 -14743.76} C_VEL
LIN {X 0,Y 326.749,Z 152.78,A -85,B 0,C 180,E1 -14746.314,E2 -14746.314} C_VEL
LIN {X 0,Y 326.772,Z 152.776,A -85,B 0,C 180,E1 -14750.092,E2 -14750.092} C_VEL
LIN {X 0,Y 326.928,Z 152.751,A -85,B 0,C 180,E1 -14753.829,E2 -14753.829} C_VEL
LIN {X 0,Y 326.996,Z 152.751,A -85,B 0,C 180,E1 -14757.536,E2 -14757.536} C_VEL
LIN {X 0,Y 327.016,Z 152.751,A -85,B 0,C 180,E1 -14761.231,E2 -14761.231} C_VEL
LIN {X 0,Y 326.739,Z 152.782,A -85,B 0,C 180,E1 -14763.7,E2 -14763.7} C_VEL
LIN {X 0,Y 326.931,Z 152.758,A -85,B 0,C 180,E1 -14766.17,E2 -14766.17} C_VEL
LIN {X 0,Y 326.772,Z 152.778,A -85,B 0,C 180,E1 -14769.907,E2 -14769.907} C_VEL
LIN {X 0,Y 326.748,Z 152.781,A -85,B 0,C 180,E1 -14773.686,E2 -14773.686} C_VEL
LIN {X 0,Y 326.653,Z 152.793,A -85,B 0,C 180,E1 -14777.53,E2 -14777.53} C_VEL
LIN {X 0,Y 326.608,Z 152.799,A -85,B 0,C 180,E1 -14781.457,E2 -14781.457} C_VEL
LIN {X 0,Y 326.644,Z 152.794,A -85,B 0,C 180,E1 -14785.488,E2 -14785.488} C_VEL
LIN {X 0,Y 326.642,Z 152.798,A -85,B 0,C 180,E1 -14788.252,E2 -14788.252} C_VEL
LIN {X 0,Y 326.585,Z 152.803,A -85,B 0,C 180,E1 -14791.096,E2 -14791.096} C_VEL
LIN {X 0,Y 326.598,Z 152.803,A -85,B 0,C 180,E1 -14794.02,E2 -14794.02} C_VEL
LIN {X 0,Y 326.619,Z 152.798,A -85,B 0,C 180,E1 -14797.24,E2 -14797.24} C_VEL
LIN {X 0,Y 326.57,Z 152.803,A -85,B 0,C 180,E1 -14801.132,E2 -14801.132} C_VEL
LIN {X 0,Y 326.521,Z 152.811,A -85,B 0,C 180,E1 -14804.744,E2 -14804.744} C_VEL
LIN {X 0,Y 326.57,Z 152.806,A -85,B 0,C 180,E1 -14808.156,E2 -14808.156} C_VEL
LIN {X 0,Y 326.618,Z 152.798,A -85,B 0,C 180,E1 -14811.393,E2 -14811.393} C_VEL
LIN {X 0,Y 326.615,Z 152.8,A -85,B 0,C 180,E1 -14814.853,E2 -14814.853} C_VEL
LIN {X 0,Y 326.657,Z 152.94,A -85,B 0,C 180,E1 -14818.463,E2 -14818.463} C_VEL
LIN {X 0,Y 329.222,Z 164.783,A -85,B 0,C 180,E1 -14821.71,E2 -14821.71} C_VEL
LIN {X 0,Y 330.631,Z 172.866,A -85,B 0,C 180,E1 -14823.83,E2 -14823.83} C_VEL
LIN {X 0,Y 329.577,Z 183.649,A -85,B 0,C 180,E1 -14826.419,E2 -14826.419} C_VEL
LIN {X 0,Y 334.372,Z 217.088,A -85,B 0,C 180,E1 -14827.491,E2 -14827.491} C_VEL
LIN {X 0,Y 335.251,Z 226.013,A -85,B 0,C 180,E1 -14827.746,E2 -14827.746} C_VEL
LIN {X 0,Y 333.948,Z 293.083,A -85,B 0,C 180,E1 -14829.2,E2 -14829.2} C_VEL
LIN {X 0,Y 333.203,Z 306.176,A -85,B 0,C 180,E1 -14829.716,E2 -14829.716} C_VEL
LIN {X 0,Y 332.258,Z 318.833,A -85,B 0,C 180,E1 -14830.461,E2 -14830.461} C_VEL
LIN {X 0,Y 331.122,Z 330.872,A -85,B 0,C 180,E1 -14831.437,E2 -14831.437} C_VEL
LIN {X 0,Y 329.825,Z 342.39,A -85,B 0,C 180,E1 -14832.645,E2 -14832.645} C_VEL
LIN {X 0,Y 328.618,Z 353.084,A -85,B 0,C 180,E1 -14834.065,E2 -14834.065} C_VEL
LIN {X 0,Y 327.526,Z 362.93,A -85,B 0,C 180,E1 -14835.715,E2 -14835.715} C_VEL
LIN {X 0,Y 326.493,Z 371.845,A -85,B 0,C 180,E1 -14837.571,E2 -14837.571} C_VEL
LIN {X 0,Y 325.747,Z 378.985,A -85,B 0,C 180,E1 -14839.434,E2 -14839.434} C_VEL
LIN {X 0,Y 325.281,Z 384.684,A -85,B 0,C 180,E1 -14841.302,E2 -14841.302} C_VEL
LIN {X 0,Y 325.045,Z 389.169,A -85,B 0,C 180,E1 -14843.172,E2 -14843.172} C_VEL
LIN {X 0,Y 324.946,Z 392.562,A -85,B 0,C 180,E1 -14845.038,E2 -14845.038} C_VEL
LIN {X 0,Y 324.967,Z 394.248,A -85,B 0,C 180,E1 -14846.281,E2 -14846.281} C_VEL
LIN {X 0,Y 324.978,Z 396.397,A -85,B 0,C 180,E1 -14848.762,E2 -14848.762} C_VEL
LIN {X 0,Y 325.041,Z 396.833,A -85,B 0,C 180,E1 -14850.001,E2 -14850.001} C_VEL
LIN {X 0,Y 324.965,Z 396.863,A -85,B 0,C 180,E1 -14851.24,E2 -14851.24} C_VEL
LIN {X 0,Y 324.933,Z 395.766,A -85,B 0,C 180,E1 -14853.721,E2 -14853.721} C_VEL
LIN {X 0,Y 324.908,Z 393.682,A -85,B 0,C 180,E1 -14855.724,E2 -14855.724} C_VEL
LIN {X 0,Y 325.196,Z 389.798,A -85,B 0,C 180,E1 -14858.076,E2 -14858.076} C_VEL
LIN {X 0,Y 325.672,Z 385.554,A -85,B 0,C 180,E1 -14859.942,E2 -14859.942} C_VEL
LIN {X 0,Y 326.523,Z 379.129,A -85,B 0,C 180,E1 -14862.115,E2 -14862.115} C_VEL
LIN {X 0,Y 327.765,Z 372.148,A -85,B 0,C 180,E1 -14863.96,E2 -14863.96} C_VEL
LIN {X 0,Y 328.959,Z 364.131,A -85,B 0,C 180,E1 -14865.668,E2 -14865.668} C_VEL
LIN {X 0,Y 330.366,Z 354.497,A -85,B 0,C 180,E1 -14867.328,E2 -14867.328} C_VEL
LIN {X 0,Y 331.955,Z 344.716,A -85,B 0,C 180,E1 -14868.677,E2 -14868.677} C_VEL
LIN {X 0,Y 333.52,Z 333.989,A -85,B 0,C 180,E1 -14869.865,E2 -14869.865} C_VEL
LIN {X 0,Y 335.023,Z 321.965,A -85,B 0,C 180,E1 -14870.894,E2 -14870.894} C_VEL
LIN {X 0,Y 336.325,Z 309.44,A -85,B 0,C 180,E1 -14871.692,E2 -14871.692} C_VEL
LIN {X 0,Y 337.287,Z 296.865,A -85,B 0,C 180,E1 -14872.25,E2 -14872.25} C_VEL
LIN {X 0,Y 337.819,Z 281.424,A -85,B 0,C 180,E1 -14872.654,E2 -14872.654} C_VEL
LIN {X 0,Y 338.956,Z 225.115,A -85,B 0,C 180,E1 -14873.857,E2 -14873.857} C_VEL
LIN {X 0,Y 335.031,Z 201.243,A -85,B 0,C 180,E1 -14874.738,E2 -14874.738} C_VEL
LIN {X 0,Y 331.499,Z 183.234,A -85,B 0,C 180,E1 -14875.479,E2 -14875.479} C_VEL
LIN {X 0,Y 332.071,Z 178.316,A -85,B 0,C 180,E1 -14876.686,E2 -14876.686} C_VEL
LIN {X 0,Y 330.961,Z 171.493,A -85,B 0,C 180,E1 -14878.542,E2 -14878.542} C_VEL
LIN {X 0,Y 328.236,Z 159.337,A -85,B 0,C 180,E1 -14882.042,E2 -14882.042} C_VEL
LIN {X 0,Y 326.629,Z 152.801,A -85,B 0,C 180,E1 -14884.064,E2 -14884.064} C_VEL
LIN {X 0,Y 326.629,Z 152.795,A -85,B 0,C 180,E1 -14887.239,E2 -14887.239} C_VEL
LIN {X 0,Y 326.58,Z 152.803,A -85,B 0,C 180,E1 -14891.131,E2 -14891.131} C_VEL
LIN {X 0,Y 326.529,Z 152.81,A -85,B 0,C 180,E1 -14894.743,E2 -14894.743} C_VEL
LIN {X 0,Y 326.564,Z 152.807,A -85,B 0,C 180,E1 -14898.152,E2 -14898.152} C_VEL
LIN {X 0,Y 326.584,Z 152.806,A -85,B 0,C 180,E1 -14901.386,E2 -14901.386} C_VEL
LIN {X 0,Y 326.619,Z 152.801,A -85,B 0,C 180,E1 -14904.852,E2 -14904.852} C_VEL
LIN {X 0,Y 326.609,Z 152.802,A -85,B 0,C 180,E1 -14907.456,E2 -14907.456} C_VEL
LIN {X 0,Y 326.617,Z 152.8,A -85,B 0,C 180,E1 -14910.337,E2 -14910.337} C_VEL
LIN {X 0,Y 326.643,Z 152.797,A -85,B 0,C 180,E1 -14914.645,E2 -14914.645} C_VEL
LIN {X 0,Y 326.61,Z 152.801,A -85,B 0,C 180,E1 -14918.543,E2 -14918.543} C_VEL
LIN {X 0,Y 326.649,Z 152.789,A -85,B 0,C 180,E1 -14921.206,E2 -14921.206} C_VEL
LIN {X 0,Y 326.718,Z 152.777,A -85,B 0,C 180,E1 -14925.465,E2 -14925.465} C_VEL
LIN {X 0,Y 326.754,Z 152.782,A -85,B 0,C 180,E1 -14928.838,E2 -14928.838} C_VEL
LIN {X 0,Y 326.913,Z 152.758,A -85,B 0,C 180,E1 -14932.589,E2 -14932.589} C_VEL
LIN {X 0,Y 326.742,Z 152.782,A -85,B 0,C 180,E1 -14935.064,E2 -14935.064} C_VEL
LIN {X 0,Y 326.986,Z 152.742,A -85,B 0,C 180,E1 -14937.536,E2 -14937.536} C_VEL
LIN {X 0,Y 327.028,Z 152.747,A -85,B 0,C 180,E1 -14941.232,E2 -14941.232} C_VEL
LIN {X 0,Y 326.739,Z 152.775,A -85,B 0,C 180,E1 -14943.7,E2 -14943.7} C_VEL
LIN {X 0,Y 326.923,Z 152.758,A -85,B 0,C 180,E1 -14946.45,E2 -14946.45} C_VEL
LIN {X 0,Y 326.785,Z 152.775,A -85,B 0,C 180,E1 -14949.907,E2 -14949.907} C_VEL
LIN {X 0,Y 326.759,Z 152.772,A -85,B 0,C 180,E1 -14953.686,E2 -14953.686} C_VEL
LIN {X 0,Y 326.666,Z 152.793,A -85,B 0,C 180,E1 -14957.53,E2 -14957.53} C_VEL
LIN {X 0,Y 326.616,Z 152.802,A -85,B 0,C 180,E1 -14961.457,E2 -14961.457} C_VEL
LIN {X 0,Y 326.64,Z 152.796,A -85,B 0,C 180,E1 -14965.488,E2 -14965.488} C_VEL
LIN {X 0,Y 326.629,Z 152.795,A -85,B 0,C 180,E1 -14968.253,E2 -14968.253} C_VEL
LIN {X 0,Y 326.577,Z 152.805,A -85,B 0,C 180,E1 -14971.097,E2 -14971.097} C_VEL
LIN {X 0,Y 326.61,Z 152.798,A -85,B 0,C 180,E1 -14974.019,E2 -14974.019} C_VEL
LIN {X 0,Y 326.63,Z 152.797,A -85,B 0,C 180,E1 -14977.238,E2 -14977.238} C_VEL
LIN {X 0,Y 326.58,Z 152.784,A -85,B 0,C 180,E1 -14981.131,E2 -14981.131} C_VEL
LIN {X 0,Y 326.531,Z 152.808,A -85,B 0,C 180,E1 -14984.743,E2 -14984.743} C_VEL
LIN {X 0,Y 326.579,Z 152.806,A -85,B 0,C 180,E1 -14988.154,E2 -14988.154} C_VEL
LIN {X 0,Y 326.601,Z 152.801,A -85,B 0,C 180,E1 -14991.387,E2 -14991.387} C_VEL
LIN {X 0,Y 326.623,Z 152.8,A -85,B 0,C 180,E1 -14994.851,E2 -14994.851} C_VEL
LIN {X 0,Y 326.651,Z 152.858,A -85,B 0,C 180,E1 -14997.87,E2 -14997.87} C_VEL
LIN {X 0,Y 327.639,Z 157.028,A -85,B 0,C 180,E1 -14999.221,E2 -14999.221} C_VEL
LIN {X 0,Y 336.899,Z 177.844,A -85,B 0,C 180,E1 -15000.55,E2 -15000.55} C_VEL
LIN {X 0,Y 339.923,Z 185.539,A -85,B 0,C 180,E1 -15000.986,E2 -15000.986} C_VEL
LIN {X 0,Y 338.11,Z 264.263,A -85,B 0,C 180,E1 -15002.686,E2 -15002.686} C_VEL
LIN {X 0,Y 337.348,Z 277.805,A -85,B 0,C 180,E1 -15003.222,E2 -15003.222} C_VEL
LIN {X 0,Y 336.321,Z 290.436,A -85,B 0,C 180,E1 -15003.97,E2 -15003.97} C_VEL
LIN {X 0,Y 335.26,Z 302.104,A -85,B 0,C 180,E1 -15004.929,E2 -15004.929} C_VEL
LIN {X 0,Y 333.868,Z 313.243,A -85,B 0,C 180,E1 -15006.094,E2 -15006.094} C_VEL
LIN {X 0,Y 332.443,Z 322.583,A -85,B 0,C 180,E1 -15007.305,E2 -15007.305} C_VEL
LIN {X 0,Y 331.055,Z 332.146,A -85,B 0,C 180,E1 -15008.844,E2 -15008.844} C_VEL
LIN {X 0,Y 329.639,Z 341.3,A -85,B 0,C 180,E1 -15010.702,E2 -15010.702} C_VEL
LIN {X 0,Y 328.256,Z 348.644,A -85,B 0,C 180,E1 -15012.557,E2 -15012.557} C_VEL
LIN {X 0,Y 327.219,Z 354.509,A -85,B 0,C 180,E1 -15014.426,E2 -15014.426} C_VEL
LIN {X 0,Y 326.389,Z 359.114,A -85,B 0,C 180,E1 -15016.298,E2 -15016.298} C_VEL
LIN {X 0,Y 325.992,Z 361.546,A -85,B 0,C 180,E1 -15017.549,E2 -15017.549} C_VEL
LIN {X 0,Y 325.596,Z 363.522,A -85,B 0,C 180,E1 -15018.797,E2 -15018.797} C_VEL
LIN {X 0,Y 325.368,Z 365.08,A -85,B 0,C 180,E1 -15020.048,E2 -15020.048} C_VEL
LIN {X 0,Y 325.223,Z 366.22,A -85,B 0,C 180,E1 -15021.299,E2 -15021.299} C_VEL
LIN {X 0,Y 325.154,Z 367.241,A -85,B 0,C 180,E1 -15023.795,E2 -15023.795} C_VEL
LIN {X 0,Y 325.077,Z 367.187,A -85,B 0,C 180,E1 -15025.038,E2 -15025.038} C_VEL
LIN {X 0,Y 325.036,Z 366.741,A -85,B 0,C 180,E1 -15026.28,E2 -15026.28} C_VEL
LIN {X 0,Y 325.116,Z 364.605,A -85,B 0,C 180,E1 -15028.76,E2 -15028.76} C_VEL
LIN {X 0,Y 325.337,Z 361.938,A -85,B 0,C 180,E1 -15030.618,E2 -15030.618} C_VEL
LIN {X 0,Y 325.66,Z 358.274,A -85,B 0,C 180,E1 -15032.473,E2 -15032.473} C_VEL
LIN {X 0,Y 326.202,Z 353.503,A -85,B 0,C 180,E1 -15034.323,E2 -15034.323} C_VEL
LIN {X 0,Y 326.967,Z 347.484,A -85,B 0,C 180,E1 -15036.168,E2 -15036.168} C_VEL
LIN {X 0,Y 327.97,Z 340.004,A -85,B 0,C 180,E1 -15038.005,E2 -15038.005} C_VEL
LIN {X 0,Y 328.892,Z 332.368,A -85,B 0,C 180,E1 -15039.531,E2 -15039.531} C_VEL
LIN {X 0,Y 329.959,Z 323.061,A -85,B 0,C 180,E1 -15041.05,E2 -15041.05} C_VEL
LIN {X 0,Y 331.144,Z 312.433,A -85,B 0,C 180,E1 -15042.442,E2 -15042.442} C_VEL
LIN {X 0,Y 332.274,Z 301.23,A -85,B 0,C 180,E1 -15043.608,E2 -15043.608} C_VEL
LIN {X 0,Y 333.137,Z 289.1,A -85,B 0,C 180,E1 -15044.585,E2 -15044.585} C_VEL
LIN {X 0,Y 333.901,Z 275.581,A -85,B 0,C 180,E1 -15045.37,E2 -15045.37} C_VEL
LIN {X 0,Y 334.432,Z 262.818,A -85,B 0,C 180,E1 -15045.853,E2 -15045.853} C_VEL
LIN {X 0,Y 336.049,Z 183.405,A -85,B 0,C 180,E1 -15047.549,E2 -15047.549} C_VEL
LIN {X 0,Y 334.1,Z 174.564,A -85,B 0,C 180,E1 -15047.875,E2 -15047.875} C_VEL
LIN {X 0,Y 327.453,Z 156.4,A -85,B 0,C 180,E1 -15048.779,E2 -15048.779} C_VEL
LIN {X 0,Y 326.699,Z 152.792,A -85,B 0,C 180,E1 -15049.897,E2 -15049.897} C_VEL
LIN {X 0,Y 326.645,Z 152.797,A -85,B 0,C 180,E1 -15054.262,E2 -15054.262} C_VEL
LIN {X 0,Y 326.659,Z 152.797,A -85,B 0,C 180,E1 -15058.102,E2 -15058.102} C_VEL
LIN {X 0,Y 326.656,Z 152.793,A -85,B 0,C 180,E1 -15059.616,E2 -15059.616} C_VEL
LIN {X 0,Y 326.032,Z 152.875,A -85,B 0,C 180,E1 -15060.645,E2 -15060.645} C_VEL
LIN {X 0,Y 323.152,Z 153.234,A -85,B 0,C 180,E1 -15062.317,E2 -15062.317} C_VEL
LIN {X 0,Y 320.685,Z 153.538,A -85,B 0,C 180,E1 -15063.673,E2 -15063.673} C_VEL
LIN {X 0,Y 319.636,Z 153.668,A -85,B 0,C 180,E1 -15064.724,E2 -15064.724} C_VEL
LIN {X 0,Y 319.558,Z 153.676,A -85,B 0,C 180,E1 -15065.08,E2 -15065.08} C_VEL
LIN {X 0,Y 319.569,Z 153.68,A -85,B 0,C 180,E1 -15068.006,E2 -15068.006} C_VEL
LIN {X 0,Y 319.521,Z 153.683,A -85,B 0,C 180,E1 -15071.595,E2 -15071.595} C_VEL
LIN {X 0,Y 319.483,Z 153.687,A -85,B 0,C 180,E1 -15075.256,E2 -15075.256} C_VEL
LIN {X 0,Y 319.522,Z 153.681,A -85,B 0,C 180,E1 -15078.71,E2 -15078.71} C_VEL
LIN {X 0,Y 319.554,Z 153.677,A -85,B 0,C 180,E1 -15082.347,E2 -15082.347} C_VEL
LIN {X 0,Y 319.552,Z 153.679,A -85,B 0,C 180,E1 -15085.122,E2 -15085.122} C_VEL
LIN {X 0,Y 319.562,Z 153.677,A -85,B 0,C 180,E1 -15089.057,E2 -15089.057} C_VEL
LIN {X 0,Y 319.589,Z 153.671,A -85,B 0,C 180,E1 -15092.496,E2 -15092.496} C_VEL
LIN {X 0,Y 319.578,Z 153.678,A -85,B 0,C 180,E1 -15095.302,E2 -15095.302} C_VEL
LIN {X 0,Y 319.558,Z 153.675,A -85,B 0,C 180,E1 -15098.045,E2 -15098.045} C_VEL
LIN {X 0,Y 319.603,Z 153.671,A -85,B 0,C 180,E1 -15102.07,E2 -15102.07} C_VEL
LIN {X 0,Y 319.722,Z 153.656,A -85,B 0,C 180,E1 -15106.007,E2 -15106.007} C_VEL
LIN {X 0,Y 319.724,Z 153.655,A -85,B 0,C 180,E1 -15109.872,E2 -15109.872} C_VEL
LIN {X 0,Y 319.886,Z 153.627,A -85,B 0,C 180,E1 -15113.693,E2 -15113.693} C_VEL
LIN {X 0,Y 319.942,Z 153.63,A -85,B 0,C 180,E1 -15117.482,E2 -15117.482} C_VEL
LIN {X 0,Y 319.986,Z 153.626,A -85,B 0,C 180,E1 -15121.258,E2 -15121.258} C_VEL
LIN {X 0,Y 319.689,Z 153.66,A -85,B 0,C 180,E1 -15123.781,E2 -15123.781} C_VEL
LIN {X 0,Y 319.888,Z 153.636,A -85,B 0,C 180,E1 -15126.307,E2 -15126.307} C_VEL
LIN {X 0,Y 319.724,Z 153.657,A -85,B 0,C 180,E1 -15130.128,E2 -15130.128} C_VEL
LIN {X 0,Y 319.721,Z 153.657,A -85,B 0,C 180,E1 -15133.993,E2 -15133.993} C_VEL
LIN {X 0,Y 319.603,Z 153.672,A -85,B 0,C 180,E1 -15137.93,E2 -15137.93} C_VEL
LIN {X 0,Y 319.558,Z 153.678,A -85,B 0,C 180,E1 -15141.955,E2 -15141.955} C_VEL
LIN {X 0,Y 319.589,Z 153.675,A -85,B 0,C 180,E1 -15146.092,E2 -15146.092} C_VEL
LIN {X 0,Y 319.577,Z 153.677,A -85,B 0,C 180,E1 -15148.935,E2 -15148.935} C_VEL
LIN {X 0,Y 319.523,Z 153.683,A -85,B 0,C 180,E1 -15151.863,E2 -15151.863} C_VEL
LIN {X 0,Y 319.571,Z 153.676,A -85,B 0,C 180,E1 -15155.544,E2 -15155.544} C_VEL
LIN {X 0,Y 319.549,Z 153.681,A -85,B 0,C 180,E1 -15158.011,E2 -15158.011} C_VEL
LIN {X 0,Y 319.518,Z 153.683,A -85,B 0,C 180,E1 -15161.598,E2 -15161.598} C_VEL
LIN {X 0,Y 319.482,Z 153.686,A -85,B 0,C 180,E1 -15165.258,E2 -15165.258} C_VEL
LIN {X 0,Y 319.523,Z 153.682,A -85,B 0,C 180,E1 -15168.713,E2 -15168.713} C_VEL
LIN {X 0,Y 319.572,Z 153.679,A -85,B 0,C 180,E1 -15172.346,E2 -15172.346} C_VEL
LIN {X 0,Y 319.556,Z 153.679,A -85,B 0,C 180,E1 -15175.125,E2 -15175.125} C_VEL
LIN {X 0,Y 319.582,Z 153.741,A -85,B 0,C 180,E1 -15178.053,E2 -15178.053} C_VEL
LIN {X 0,Y 322.11,Z 165.327,A -85,B 0,C 180,E1 -15181.316,E2 -15181.316} C_VEL
LIN {X 0,Y 323.642,Z 173.751,A -85,B 0,C 180,E1 -15183.585,E2 -15183.585} C_VEL
LIN {X 0,Y 322.774,Z 183.544,A -85,B 0,C 180,E1 -15185.949,E2 -15185.949} C_VEL
LIN {X 0,Y 326.98,Z 212.336,A -85,B 0,C 180,E1 -15186.906,E2 -15186.906} C_VEL
LIN {X 0,Y 328.593,Z 226.393,A -85,B 0,C 180,E1 -15187.333,E2 -15187.333} C_VEL
LIN {X 0,Y 327.209,Z 292.585,A -85,B 0,C 180,E1 -15188.792,E2 -15188.792} C_VEL
LIN {X 0,Y 326.499,Z 305.746,A -85,B 0,C 180,E1 -15189.321,E2 -15189.321} C_VEL
LIN {X 0,Y 325.549,Z 317.863,A -85,B 0,C 180,E1 -15190.042,E2 -15190.042} C_VEL
LIN {X 0,Y 324.347,Z 330.091,A -85,B 0,C 180,E1 -15191.035,E2 -15191.035} C_VEL
LIN {X 0,Y 323.014,Z 341.694,A -85,B 0,C 180,E1 -15192.267,E2 -15192.267} C_VEL
LIN {X 0,Y 321.749,Z 352.267,A -85,B 0,C 180,E1 -15193.685,E2 -15193.685} C_VEL
LIN {X 0,Y 320.863,Z 360.709,A -85,B 0,C 180,E1 -15195.088,E2 -15195.088} C_VEL
LIN {X 0,Y 319.88,Z 368.585,A -85,B 0,C 180,E1 -15196.664,E2 -15196.664} C_VEL
LIN {X 0,Y 318.909,Z 376.269,A -85,B 0,C 180,E1 -15198.562,E2 -15198.562} C_VEL
LIN {X 0,Y 318.333,Z 382.457,A -85,B 0,C 180,E1 -15200.47,E2 -15200.47} C_VEL
LIN {X 0,Y 318.01,Z 387.365,A -85,B 0,C 180,E1 -15202.381,E2 -15202.381} C_VEL
LIN {X 0,Y 317.906,Z 390.927,A -85,B 0,C 180,E1 -15204.169,E2 -15204.169} C_VEL
LIN {X 0,Y 317.893,Z 393.873,A -85,B 0,C 180,E1 -15206.198,E2 -15206.198} C_VEL
LIN {X 0,Y 317.882,Z 396.048,A -85,B 0,C 180,E1 -15208.734,E2 -15208.734} C_VEL
LIN {X 0,Y 317.948,Z 396.503,A -85,B 0,C 180,E1 -15210.001,E2 -15210.001} C_VEL
LIN {X 0,Y 317.868,Z 396.545,A -85,B 0,C 180,E1 -15211.268,E2 -15211.268} C_VEL
LIN {X 0,Y 317.835,Z 395.47,A -85,B 0,C 180,E1 -15213.805,E2 -15213.805} C_VEL
LIN {X 0,Y 317.825,Z 393.601,A -85,B 0,C 180,E1 -15215.688,E2 -15215.688} C_VEL
LIN {X 0,Y 318.015,Z 390.729,A -85,B 0,C 180,E1 -15217.621,E2 -15217.621} C_VEL
LIN {X 0,Y 318.447,Z 386.869,A -85,B 0,C 180,E1 -15219.529,E2 -15219.529} C_VEL
LIN {X 0,Y 319.096,Z 381.894,A -85,B 0,C 180,E1 -15221.434,E2 -15221.434} C_VEL
LIN {X 0,Y 320.165,Z 375.661,A -85,B 0,C 180,E1 -15223.327,E2 -15223.327} C_VEL
LIN {X 0,Y 321.214,Z 369.303,A -85,B 0,C 180,E1 -15224.898,E2 -15224.898} C_VEL
LIN {X 0,Y 322.696,Z 359.996,A -85,B 0,C 180,E1 -15226.773,E2 -15226.773} C_VEL
LIN {X 0,Y 324.31,Z 350.365,A -85,B 0,C 180,E1 -15228.315,E2 -15228.315} C_VEL
LIN {X 0,Y 326.023,Z 339.692,A -85,B 0,C 180,E1 -15229.684,E2 -15229.684} C_VEL
LIN {X 0,Y 327.497,Z 329.381,A -85,B 0,C 180,E1 -15230.738,E2 -15230.738} C_VEL
LIN {X 0,Y 329.014,Z 317.069,A -85,B 0,C 180,E1 -15231.705,E2 -15231.705} C_VEL
LIN {X 0,Y 330.275,Z 304.125,A -85,B 0,C 180,E1 -15232.44,E2 -15232.44} C_VEL
LIN {X 0,Y 331.125,Z 291.482,A -85,B 0,C 180,E1 -15232.917,E2 -15232.917} C_VEL
LIN {X 0,Y 332.607,Z 226.309,A -85,B 0,C 180,E1 -15234.353,E2 -15234.353} C_VEL
LIN {X 0,Y 328.714,Z 202.564,A -85,B 0,C 180,E1 -15235.256,E2 -15235.256} C_VEL
LIN {X 0,Y 324.865,Z 182.87,A -85,B 0,C 180,E1 -15236.096,E2 -15236.096} C_VEL
LIN {X 0,Y 325.187,Z 179.338,A -85,B 0,C 180,E1 -15236.992,E2 -15236.992} C_VEL
LIN {X 0,Y 323.836,Z 171.768,A -85,B 0,C 180,E1 -15239.118,E2 -15239.118} C_VEL
LIN {X 0,Y 321.313,Z 160.683,A -85,B 0,C 180,E1 -15242.404,E2 -15242.404} C_VEL
LIN {X 0,Y 319.6,Z 153.673,A -85,B 0,C 180,E1 -15244.589,E2 -15244.589} C_VEL
LIN {X 0,Y 319.575,Z 153.677,A -85,B 0,C 180,E1 -15248.009,E2 -15248.009} C_VEL
LIN {X 0,Y 319.528,Z 153.683,A -85,B 0,C 180,E1 -15251.597,E2 -15251.597} C_VEL
LIN {X 0,Y 319.49,Z 153.689,A -85,B 0,C 180,E1 -15255.257,E2 -15255.257} C_VEL
LIN {X 0,Y 319.507,Z 153.686,A -85,B 0,C 180,E1 -15258.408,E2 -15258.408} C_VEL
LIN {X 0,Y 319.533,Z 153.683,A -85,B 0,C 180,E1 -15261.986,E2 -15261.986} C_VEL
LIN {X 0,Y 319.56,Z 153.68,A -85,B 0,C 180,E1 -15265.123,E2 -15265.123} C_VEL
LIN {X 0,Y 319.526,Z 153.683,A -85,B 0,C 180,E1 -15268.138,E2 -15268.138} C_VEL
LIN {X 0,Y 319.572,Z 153.675,A -85,B 0,C 180,E1 -15271.604,E2 -15271.604} C_VEL
LIN {X 0,Y 319.573,Z 153.677,A -85,B 0,C 180,E1 -15275.301,E2 -15275.301} C_VEL
LIN {X 0,Y 319.564,Z 153.678,A -85,B 0,C 180,E1 -15278.045,E2 -15278.045} C_VEL
LIN {X 0,Y 319.587,Z 153.671,A -85,B 0,C 180,E1 -15282.069,E2 -15282.069} C_VEL
LIN {X 0,Y 319.701,Z 153.65,A -85,B 0,C 180,E1 -15286.006,E2 -15286.006} C_VEL
LIN {X 0,Y 319.734,Z 153.656,A -85,B 0,C 180,E1 -15289.872,E2 -15289.872} C_VEL
LIN {X 0,Y 319.897,Z 153.635,A -85,B 0,C 180,E1 -15293.694,E2 -15293.694} C_VEL
LIN {X 0,Y 319.996,Z 153.622,A -85,B 0,C 180,E1 -15298.742,E2 -15298.742} C_VEL
LIN {X 0,Y 319.949,Z 153.618,A -85,B 0,C 180,E1 -15302.518,E2 -15302.518} C_VEL
LIN {X 0,Y 319.889,Z 153.635,A -85,B 0,C 180,E1 -15306.431,E2 -15306.431} C_VEL
LIN {X 0,Y 319.737,Z 153.655,A -85,B 0,C 180,E1 -15310.128,E2 -15310.128} C_VEL
LIN {X 0,Y 319.733,Z 153.645,A -85,B 0,C 180,E1 -15313.992,E2 -15313.992} C_VEL
LIN {X 0,Y 319.616,Z 153.668,A -85,B 0,C 180,E1 -15317.93,E2 -15317.93} C_VEL
LIN {X 0,Y 319.568,Z 153.677,A -85,B 0,C 180,E1 -15321.955,E2 -15321.955} C_VEL
LIN {X 0,Y 319.576,Z 153.675,A -85,B 0,C 180,E1 -15326.093,E2 -15326.093} C_VEL
LIN {X 0,Y 319.56,Z 153.673,A -85,B 0,C 180,E1 -15328.937,E2 -15328.937} C_VEL
LIN {X 0,Y 319.527,Z 153.68,A -85,B 0,C 180,E1 -15331.863,E2 -15331.863} C_VEL
LIN {X 0,Y 319.582,Z 153.673,A -85,B 0,C 180,E1 -15335.543,E2 -15335.543} C_VEL
LIN {X 0,Y 319.56,Z 153.678,A -85,B 0,C 180,E1 -15338.01,E2 -15338.01} C_VEL
LIN {X 0,Y 319.529,Z 153.663,A -85,B 0,C 180,E1 -15341.597,E2 -15341.597} C_VEL
LIN {X 0,Y 319.491,Z 153.684,A -85,B 0,C 180,E1 -15345.257,E2 -15345.257} C_VEL
LIN {X 0,Y 319.531,Z 153.684,A -85,B 0,C 180,E1 -15348.711,E2 -15348.711} C_VEL
LIN {X 0,Y 319.558,Z 153.68,A -85,B 0,C 180,E1 -15352.349,E2 -15352.349} C_VEL
LIN {X 0,Y 319.564,Z 153.679,A -85,B 0,C 180,E1 -15355.123,E2 -15355.123} C_VEL
LIN {X 0,Y 319.576,Z 153.695,A -85,B 0,C 180,E1 -15357.309,E2 -15357.309} C_VEL
LIN {X 0,Y 320.49,Z 157.445,A -85,B 0,C 180,E1 -15358.543,E2 -15358.543} C_VEL
LIN {X 0,Y 329.198,Z 176.666,A -85,B 0,C 180,E1 -15359.841,E2 -15359.841} C_VEL
LIN {X 0,Y 333.609,Z 187.488,A -85,B 0,C 180,E1 -15360.492,E2 -15360.492} C_VEL
LIN {X 0,Y 331.684,Z 264.628,A -85,B 0,C 180,E1 -15362.183,E2 -15362.183} C_VEL
LIN {X 0,Y 330.917,Z 277.637,A -85,B 0,C 180,E1 -15362.702,E2 -15362.702} C_VEL
LIN {X 0,Y 329.891,Z 289.834,A -85,B 0,C 180,E1 -15363.423,E2 -15363.423} C_VEL
LIN {X 0,Y 328.748,Z 302.024,A -85,B 0,C 180,E1 -15364.423,E2 -15364.423} C_VEL
LIN {X 0,Y 327.344,Z 313.034,A -85,B 0,C 180,E1 -15365.587,E2 -15365.587} C_VEL
LIN {X 0,Y 325.677,Z 323.539,A -85,B 0,C 180,E1 -15366.974,E2 -15366.974} C_VEL
LIN {X 0,Y 324.374,Z 332.104,A -85,B 0,C 180,E1 -15368.387,E2 -15368.387} C_VEL
LIN {X 0,Y 323.138,Z 339.972,A -85,B 0,C 180,E1 -15369.967,E2 -15369.967} C_VEL
LIN {X 0,Y 321.641,Z 347.623,A -85,B 0,C 180,E1 -15371.857,E2 -15371.857} C_VEL
LIN {X 0,Y 320.304,Z 354.647,A -85,B 0,C 180,E1 -15374.08,E2 -15374.08} C_VEL
LIN {X 0,Y 319.429,Z 359.292,A -85,B 0,C 180,E1 -15375.993,E2 -15375.993} C_VEL
LIN {X 0,Y 319.004,Z 361.761,A -85,B 0,C 180,E1 -15377.272,E2 -15377.272} C_VEL
LIN {X 0,Y 318.574,Z 363.756,A -85,B 0,C 180,E1 -15378.547,E2 -15378.547} C_VEL
LIN {X 0,Y 318.327,Z 365.33,A -85,B 0,C 180,E1 -15379.826,E2 -15379.826} C_VEL
LIN {X 0,Y 318.149,Z 366.498,A -85,B 0,C 180,E1 -15381.104,E2 -15381.104} C_VEL
LIN {X 0,Y 318.064,Z 367.558,A -85,B 0,C 180,E1 -15383.656,E2 -15383.656} C_VEL
LIN {X 0,Y 318.005,Z 367.519,A -85,B 0,C 180,E1 -15384.927,E2 -15384.927} C_VEL
LIN {X 0,Y 317.963,Z 367.098,A -85,B 0,C 180,E1 -15386.197,E2 -15386.197} C_VEL
LIN {X 0,Y 318.019,Z 365.004,A -85,B 0,C 180,E1 -15388.733,E2 -15388.733} C_VEL
LIN {X 0,Y 318.267,Z 362.37,A -85,B 0,C 180,E1 -15390.631,E2 -15390.631} C_VEL
LIN {X 0,Y 318.603,Z 358.742,A -85,B 0,C 180,E1 -15392.527,E2 -15392.527} C_VEL
LIN {X 0,Y 319.154,Z 354.011,A -85,B 0,C 180,E1 -15394.419,E2 -15394.419} C_VEL
LIN {X 0,Y 319.939,Z 348.036,A -85,B 0,C 180,E1 -15396.304,E2 -15396.304} C_VEL
LIN {X 0,Y 320.976,Z 340.604,A -85,B 0,C 180,E1 -15398.181,E2 -15398.181} C_VEL
LIN {X 0,Y 321.93,Z 333.025,A -85,B 0,C 180,E1 -15399.739,E2 -15399.739} C_VEL
LIN {X 0,Y 323.036,Z 323.821,A -85,B 0,C 180,E1 -15401.29,E2 -15401.29} C_VEL
LIN {X 0,Y 324.241,Z 313.573,A -85,B 0,C 180,E1 -15402.676,E2 -15402.676} C_VEL
LIN {X 0,Y 325.421,Z 302.201,A -85,B 0,C 180,E1 -15403.901,E2 -15403.901} C_VEL
LIN {X 0,Y 326.352,Z 290.339,A -85,B 0,C 180,E1 -15404.895,E2 -15404.895} C_VEL
LIN {X 0,Y 327.08,Z 277.908,A -85,B 0,C 180,E1 -15405.659,E2 -15405.659} C_VEL
LIN {X 0,Y 327.648,Z 265.097,A -85,B 0,C 180,E1 -15406.19,E2 -15406.19} C_VEL
LIN {X 0,Y 328.718,Z 218.302,A -85,B 0,C 180,E1 -15407.235,E2 -15407.235} C_VEL
LIN {X 0,Y 329.283,Z 183.825,A -85,B 0,C 180,E1 -15407.987,E2 -15407.987} C_VEL
LIN {X 0,Y 327.682,Z 176.63,A -85,B 0,C 180,E1 -15408.262,E2 -15408.262} C_VEL
LIN {X 0,Y 320.321,Z 156.728,A -85,B 0,C 180,E1 -15409.288,E2 -15409.288} C_VEL
LIN {X 0,Y 319.605,Z 153.676,A -85,B 0,C 180,E1 -15410.262,E2 -15410.262} C_VEL
LIN {X 0,Y 319.559,Z 153.678,A -85,B 0,C 180,E1 -15413.319,E2 -15413.319} C_VEL
LIN {X 0,Y 319.634,Z 153.672,A -85,B 0,C 180,E1 -15416.086,E2 -15416.086} C_VEL
LIN {X 0,Y 319.563,Z 153.675,A -85,B 0,C 180,E1 -15419.615,E2 -15419.615} C_VEL
LIN {X 0,Y 319.573,Z 153.675,A -85,B 0,C 180,E1 -15423.351,E2 -15423.351} C_VEL
LIN {X 0,Y 319.558,Z 153.676,A -85,B 0,C 180,E1 -15425.08,E2 -15425.08} C_VEL
LIN {X 0,Y 318.906,Z 153.762,A -85,B 0,C 180,E1 -15426.132,E2 -15426.132} C_VEL
LIN {X 0,Y 316.044,Z 154.118,A -85,B 0,C 180,E1 -15427.844,E2 -15427.844} C_VEL
LIN {X 0,Y 313.609,Z 154.421,A -85,B 0,C 180,E1 -15429.232,E2 -15429.232} C_VEL
LIN {X 0,Y 312.567,Z 154.55,A -85,B 0,C 180,E1 -15430.307,E2 -15430.307} C_VEL
LIN {X 0,Y 312.485,Z 154.557,A -85,B 0,C 180,E1 -15430.671,E2 -15430.671} C_VEL
LIN {X 0,Y 312.446,Z 154.566,A -85,B 0,C 180,E1 -15434.208,E2 -15434.208} C_VEL
LIN {X 0,Y 312.478,Z 154.562,A -85,B 0,C 180,E1 -15437.917,E2 -15437.917} C_VEL
LIN {X 0,Y 312.528,Z 154.555,A -85,B 0,C 180,E1 -15441.909,E2 -15441.909} C_VEL
LIN {X 0,Y 312.499,Z 154.559,A -85,B 0,C 180,E1 -15445.789,E2 -15445.789} C_VEL
LIN {X 0,Y 312.515,Z 154.554,A -85,B 0,C 180,E1 -15448.853,E2 -15448.853} C_VEL
LIN {X 0,Y 312.561,Z 154.549,A -85,B 0,C 180,E1 -15451.823,E2 -15451.823} C_VEL
LIN {X 0,Y 312.552,Z 154.55,A -85,B 0,C 180,E1 -15454.708,E2 -15454.708} C_VEL
LIN {X 0,Y 312.555,Z 154.551,A -85,B 0,C 180,E1 -15457.526,E2 -15457.526} C_VEL
LIN {X 0,Y 312.557,Z 154.552,A -85,B 0,C 180,E1 -15461.651,E2 -15461.651} C_VEL
LIN {X 0,Y 312.675,Z 154.536,A -85,B 0,C 180,E1 -15465.685,E2 -15465.685} C_VEL
LIN {X 0,Y 312.675,Z 154.534,A -85,B 0,C 180,E1 -15469.641,E2 -15469.641} C_VEL
LIN {X 0,Y 312.784,Z 154.514,A -85,B 0,C 180,E1 -15472.252,E2 -15472.252} C_VEL
LIN {X 0,Y 312.674,Z 154.525,A -85,B 0,C 180,E1 -15474.842,E2 -15474.842} C_VEL
LIN {X 0,Y 312.955,Z 154.5,A -85,B 0,C 180,E1 -15478.713,E2 -15478.713} C_VEL
LIN {X 0,Y 312.892,Z 154.508,A -85,B 0,C 180,E1 -15482.575,E2 -15482.575} C_VEL
LIN {X 0,Y 312.83,Z 154.516,A -85,B 0,C 180,E1 -15486.45,E2 -15486.45} C_VEL
LIN {X 0,Y 312.74,Z 154.53,A -85,B 0,C 180,E1 -15489.05,E2 -15489.05} C_VEL
LIN {X 0,Y 312.624,Z 154.545,A -85,B 0,C 180,E1 -15492.991,E2 -15492.991} C_VEL
LIN {X 0,Y 312.611,Z 154.542,A -85,B 0,C 180,E1 -15495.651,E2 -15495.651} C_VEL
LIN {X 0,Y 312.529,Z 154.553,A -85,B 0,C 180,E1 -15499.713,E2 -15499.713} C_VEL
LIN {X 0,Y 312.516,Z 154.559,A -85,B 0,C 180,E1 -15502.781,E2 -15502.781} C_VEL
LIN {X 0,Y 312.565,Z 154.549,A -85,B 0,C 180,E1 -15505.925,E2 -15505.925} C_VEL
LIN {X 0,Y 312.535,Z 154.553,A -85,B 0,C 180,E1 -15509.651,E2 -15509.651} C_VEL
LIN {X 0,Y 312.511,Z 154.556,A -85,B 0,C 180,E1 -15513.69,E2 -15513.69} C_VEL
LIN {X 0,Y 312.517,Z 154.555,A -85,B 0,C 180,E1 -15517.386,E2 -15517.386} C_VEL
LIN {X 0,Y 312.483,Z 154.56,A -85,B 0,C 180,E1 -15520.71,E2 -15520.71} C_VEL
LIN {X 0,Y 312.445,Z 154.568,A -85,B 0,C 180,E1 -15524.211,E2 -15524.211} C_VEL
LIN {X 0,Y 312.478,Z 154.56,A -85,B 0,C 180,E1 -15527.92,E2 -15527.92} C_VEL
LIN {X 0,Y 312.529,Z 154.557,A -85,B 0,C 180,E1 -15531.912,E2 -15531.912} C_VEL
LIN {X 0,Y 312.502,Z 154.562,A -85,B 0,C 180,E1 -15535.791,E2 -15535.791} C_VEL
LIN {X 0,Y 312.555,Z 154.706,A -85,B 0,C 180,E1 -15537.674,E2 -15537.674} C_VEL
LIN {X 0,Y 315.082,Z 166.134,A -85,B 0,C 180,E1 -15540.98,E2 -15540.98} C_VEL
LIN {X 0,Y 316.589,Z 174.165,A -85,B 0,C 180,E1 -15543.203,E2 -15543.203} C_VEL
LIN {X 0,Y 316.456,Z 178.584,A -85,B 0,C 180,E1 -15544.339,E2 -15544.339} C_VEL
LIN {X 0,Y 315.926,Z 182.973,A -85,B 0,C 180,E1 -15545.436,E2 -15545.436} C_VEL
LIN {X 0,Y 320.177,Z 211.743,A -85,B 0,C 180,E1 -15546.43,E2 -15546.43} C_VEL
LIN {X 0,Y 321.943,Z 226.856,A -85,B 0,C 180,E1 -15546.906,E2 -15546.906} C_VEL
LIN {X 0,Y 320.523,Z 292.086,A -85,B 0,C 180,E1 -15548.37,E2 -15548.37} C_VEL
LIN {X 0,Y 319.81,Z 305.31,A -85,B 0,C 180,E1 -15548.911,E2 -15548.911} C_VEL
LIN {X 0,Y 318.745,Z 318.02,A -85,B 0,C 180,E1 -15549.681,E2 -15549.681} C_VEL
LIN {X 0,Y 317.594,Z 329.308,A -85,B 0,C 180,E1 -15550.615,E2 -15550.615} C_VEL
LIN {X 0,Y 316.198,Z 340.994,A -85,B 0,C 180,E1 -15551.872,E2 -15551.872} C_VEL
LIN {X 0,Y 314.912,Z 351.487,A -85,B 0,C 180,E1 -15553.298,E2 -15553.298} C_VEL
LIN {X 0,Y 313.948,Z 360.127,A -85,B 0,C 180,E1 -15554.751,E2 -15554.751} C_VEL
LIN {X 0,Y 312.926,Z 368.054,A -85,B 0,C 180,E1 -15556.361,E2 -15556.361} C_VEL
LIN {X 0,Y 311.914,Z 375.784,A -85,B 0,C 180,E1 -15558.301,E2 -15558.301} C_VEL
LIN {X 0,Y 311.299,Z 382.002,A -85,B 0,C 180,E1 -15560.253,E2 -15560.253} C_VEL
LIN {X 0,Y 310.957,Z 386.939,A -85,B 0,C 180,E1 -15562.208,E2 -15562.208} C_VEL
LIN {X 0,Y 310.821,Z 390.807,A -85,B 0,C 180,E1 -15564.204,E2 -15564.204} C_VEL
LIN {X 0,Y 310.798,Z 393.497,A -85,B 0,C 180,E1 -15566.111,E2 -15566.111} C_VEL
LIN {X 0,Y 310.768,Z 394.795,A -85,B 0,C 180,E1 -15567.409,E2 -15567.409} C_VEL
LIN {X 0,Y 310.789,Z 395.696,A -85,B 0,C 180,E1 -15568.705,E2 -15568.705} C_VEL
LIN {X 0,Y 310.854,Z 396.174,A -85,B 0,C 180,E1 -15570.001,E2 -15570.001} C_VEL
LIN {X 0,Y 310.775,Z 396.226,A -85,B 0,C 180,E1 -15571.297,E2 -15571.297} C_VEL
LIN {X 0,Y 310.742,Z 395.174,A -85,B 0,C 180,E1 -15573.892,E2 -15573.892} C_VEL
LIN {X 0,Y 310.724,Z 393.558,A -85,B 0,C 180,E1 -15575.615,E2 -15575.615} C_VEL
LIN {X 0,Y 310.969,Z 390.48,A -85,B 0,C 180,E1 -15577.795,E2 -15577.795} C_VEL
LIN {X 0,Y 311.402,Z 386.645,A -85,B 0,C 180,E1 -15579.746,E2 -15579.746} C_VEL
LIN {X 0,Y 312.097,Z 381.697,A -85,B 0,C 180,E1 -15581.694,E2 -15581.694} C_VEL
LIN {X 0,Y 313.236,Z 375.495,A -85,B 0,C 180,E1 -15583.627,E2 -15583.627} C_VEL
LIN {X 0,Y 314.575,Z 367.793,A -85,B 0,C 180,E1 -15585.552,E2 -15585.552} C_VEL
LIN {X 0,Y 315.891,Z 359.927,A -85,B 0,C 180,E1 -15587.146,E2 -15587.146} C_VEL
LIN {X 0,Y 317.555,Z 350.349,A -85,B 0,C 180,E1 -15588.719,E2 -15588.719} C_VEL
LIN {X 0,Y 319.361,Z 339.741,A -85,B 0,C 180,E1 -15590.113,E2 -15590.113} C_VEL
LIN {X 0,Y 321.096,Z 327.863,A -85,B 0,C 180,E1 -15591.34,E2 -15591.34} C_VEL
LIN {X 0,Y 322.715,Z 315.142,A -85,B 0,C 180,E1 -15592.319,E2 -15592.319} C_VEL
LIN {X 0,Y 323.925,Z 302.453,A -85,B 0,C 180,E1 -15593.028,E2 -15593.028} C_VEL
LIN {X 0,Y 324.706,Z 290.038,A -85,B 0,C 180,E1 -15593.48,E2 -15593.48} C_VEL
LIN {X 0,Y 326.193,Z 226.882,A -85,B 0,C 180,E1 -15594.893,E2 -15594.893} C_VEL
LIN {X 0,Y 322.451,Z 204.11,A -85,B 0,C 180,E1 -15595.786,E2 -15595.786} C_VEL
LIN {X 0,Y 318.261,Z 182.506,A -85,B 0,C 180,E1 -15596.741,E2 -15596.741} C_VEL
LIN {X 0,Y 317.977,Z 178.431,A -85,B 0,C 180,E1 -15597.86,E2 -15597.86} C_VEL
LIN {X 0,Y 315.618,Z 167.396,A -85,B 0,C 180,E1 -15601.126,E2 -15601.126} C_VEL
LIN {X 0,Y 313.033,Z 156.533,A -85,B 0,C 180,E1 -15604.535,E2 -15604.535} C_VEL
LIN {X 0,Y 312.536,Z 154.554,A -85,B 0,C 180,E1 -15605.187,E2 -15605.187} C_VEL
LIN {X 0,Y 312.51,Z 154.551,A -85,B 0,C 180,E1 -15609.028,E2 -15609.028} C_VEL
LIN {X 0,Y 312.492,Z 154.556,A -85,B 0,C 180,E1 -15612.432,E2 -15612.432} C_VEL
LIN {X 0,Y 312.46,Z 154.564,A -85,B 0,C 180,E1 -15616.035,E2 -15616.035} C_VEL
LIN {X 0,Y 312.457,Z 154.565,A -85,B 0,C 180,E1 -15619.886,E2 -15619.886} C_VEL
LIN {X 0,Y 312.535,Z 154.555,A -85,B 0,C 180,E1 -15624.051,E2 -15624.051} C_VEL
LIN {X 0,Y 312.503,Z 154.559,A -85,B 0,C 180,E1 -15627.334,E2 -15627.334} C_VEL
LIN {X 0,Y 312.508,Z 154.556,A -85,B 0,C 180,E1 -15631.292,E2 -15631.292} C_VEL
LIN {X 0,Y 312.548,Z 154.553,A -85,B 0,C 180,E1 -15634.708,E2 -15634.708} C_VEL
LIN {X 0,Y 312.542,Z 154.552,A -85,B 0,C 180,E1 -15637.526,E2 -15637.526} C_VEL
LIN {X 0,Y 312.552,Z 154.546,A -85,B 0,C 180,E1 -15641.651,E2 -15641.651} C_VEL
LIN {X 0,Y 312.643,Z 154.529,A -85,B 0,C 180,E1 -15645.684,E2 -15645.684} C_VEL
LIN {X 0,Y 312.684,Z 154.534,A -85,B 0,C 180,E1 -15649.641,E2 -15649.641} C_VEL
LIN {X 0,Y 312.839,Z 154.514,A -85,B 0,C 180,E1 -15653.551,E2 -15653.551} C_VEL
LIN {X 0,Y 312.964,Z 154.498,A -85,B 0,C 180,E1 -15658.713,E2 -15658.713} C_VEL
LIN {X 0,Y 312.966,Z 154.499,A -85,B 0,C 180,E1 -15661.287,E2 -15661.287} C_VEL
LIN {X 0,Y 312.687,Z 154.533,A -85,B 0,C 180,E1 -15665.158,E2 -15665.158} C_VEL
LIN {X 0,Y 312.797,Z 154.512,A -85,B 0,C 180,E1 -15667.748,E2 -15667.748} C_VEL
LIN {X 0,Y 312.665,Z 154.539,A -85,B 0,C 180,E1 -15671.672,E2 -15671.672} C_VEL
LIN {X 0,Y 312.67,Z 154.526,A -85,B 0,C 180,E1 -15674.865,E2 -15674.865} C_VEL
LIN {X 0,Y 312.55,Z 154.543,A -85,B 0,C 180,E1 -15679.193,E2 -15679.193} C_VEL
LIN {X 0,Y 312.525,Z 154.556,A -85,B 0,C 180,E1 -15682.779,E2 -15682.779} C_VEL
LIN {X 0,Y 312.535,Z 154.552,A -85,B 0,C 180,E1 -15685.909,E2 -15685.909} C_VEL
LIN {X 0,Y 312.506,Z 154.555,A -85,B 0,C 180,E1 -15689.654,E2 -15689.654} C_VEL
LIN {X 0,Y 312.523,Z 154.553,A -85,B 0,C 180,E1 -15693.689,E2 -15693.689} C_VEL
LIN {X 0,Y 312.529,Z 154.553,A -85,B 0,C 180,E1 -15697.385,E2 -15697.385} C_VEL
LIN {X 0,Y 312.493,Z 154.538,A -85,B 0,C 180,E1 -15700.709,E2 -15700.709} C_VEL
LIN {X 0,Y 312.455,Z 154.566,A -85,B 0,C 180,E1 -15704.209,E2 -15704.209} C_VEL
LIN {X 0,Y 312.487,Z 154.559,A -85,B 0,C 180,E1 -15707.919,E2 -15707.919} C_VEL
LIN {X 0,Y 312.502,Z 154.558,A -85,B 0,C 180,E1 -15710.971,E2 -15710.971} C_VEL
LIN {X 0,Y 312.536,Z 154.554,A -85,B 0,C 180,E1 -15714.22,E2 -15714.22} C_VEL
LIN {X 0,Y 312.539,Z 154.577,A -85,B 0,C 180,E1 -15716.735,E2 -15716.735} C_VEL
LIN {X 0,Y 313.379,Z 157.966,A -85,B 0,C 180,E1 -15717.835,E2 -15717.835} C_VEL
LIN {X 0,Y 322.636,Z 177.974,A -85,B 0,C 180,E1 -15719.262,E2 -15719.262} C_VEL
LIN {X 0,Y 327.288,Z 189.441,A -85,B 0,C 180,E1 -15719.976,E2 -15719.976} C_VEL
LIN {X 0,Y 325.268,Z 265.05,A -85,B 0,C 180,E1 -15721.661,E2 -15721.661} C_VEL
LIN {X 0,Y 324.467,Z 278.242,A -85,B 0,C 180,E1 -15722.2,E2 -15722.2} C_VEL
LIN {X 0,Y 323.324,Z 291.113,A -85,B 0,C 180,E1 -15722.985,E2 -15722.985} C_VEL
LIN {X 0,Y 322.135,Z 303.053,A -85,B 0,C 180,E1 -15724.007,E2 -15724.007} C_VEL
LIN {X 0,Y 320.637,Z 314.124,A -85,B 0,C 180,E1 -15725.215,E2 -15725.215} C_VEL
LIN {X 0,Y 319.077,Z 323.423,A -85,B 0,C 180,E1 -15726.47,E2 -15726.47} C_VEL
LIN {X 0,Y 317.721,Z 332.063,A -85,B 0,C 180,E1 -15727.91,E2 -15727.91} C_VEL
LIN {X 0,Y 316.393,Z 339.995,A -85,B 0,C 180,E1 -15729.521,E2 -15729.521} C_VEL
LIN {X 0,Y 314.837,Z 347.719,A -85,B 0,C 180,E1 -15731.451,E2 -15731.451} C_VEL
LIN {X 0,Y 313.408,Z 354.787,A -85,B 0,C 180,E1 -15733.721,E2 -15733.721} C_VEL
LIN {X 0,Y 312.482,Z 359.471,A -85,B 0,C 180,E1 -15735.675,E2 -15735.675} C_VEL
LIN {X 0,Y 311.792,Z 363.035,A -85,B 0,C 180,E1 -15737.634,E2 -15737.634} C_VEL
LIN {X 0,Y 311.299,Z 365.581,A -85,B 0,C 180,E1 -15739.594,E2 -15739.594} C_VEL
LIN {X 0,Y 311.091,Z 366.771,A -85,B 0,C 180,E1 -15740.9,E2 -15740.9} C_VEL
LIN {X 0,Y 310.992,Z 367.523,A -85,B 0,C 180,E1 -15742.206,E2 -15742.206} C_VEL
LIN {X 0,Y 311.014,Z 367.913,A -85,B 0,C 180,E1 -15743.868,E2 -15743.868} C_VEL
LIN {X 0,Y 310.893,Z 367.45,A -85,B 0,C 180,E1 -15746.11,E2 -15746.11} C_VEL
LIN {X 0,Y 310.845,Z 366.631,A -85,B 0,C 180,E1 -15747.407,E2 -15747.407} C_VEL
LIN {X 0,Y 311.094,Z 363.777,A -85,B 0,C 180,E1 -15749.999,E2 -15749.999} C_VEL
LIN {X 0,Y 311.398,Z 360.521,A -85,B 0,C 180,E1 -15751.939,E2 -15751.939} C_VEL
LIN {X 0,Y 311.895,Z 356.21,A -85,B 0,C 180,E1 -15753.875,E2 -15753.875} C_VEL
LIN {X 0,Y 312.585,Z 350.723,A -85,B 0,C 180,E1 -15755.806,E2 -15755.806} C_VEL
LIN {X 0,Y 313.526,Z 343.877,A -85,B 0,C 180,E1 -15757.728,E2 -15757.728} C_VEL
LIN {X 0,Y 314.831,Z 335.285,A -85,B 0,C 180,E1 -15759.637,E2 -15759.637} C_VEL
LIN {X 0,Y 315.642,Z 328.442,A -85,B 0,C 180,E1 -15760.908,E2 -15760.908} C_VEL
LIN {X 0,Y 316.824,Z 319.178,A -85,B 0,C 180,E1 -15762.328,E2 -15762.328} C_VEL
LIN {X 0,Y 318.101,Z 307.709,A -85,B 0,C 180,E1 -15763.738,E2 -15763.738} C_VEL
LIN {X 0,Y 319.214,Z 296.386,A -85,B 0,C 180,E1 -15764.828,E2 -15764.828} C_VEL
LIN {X 0,Y 320.007,Z 284.745,A -85,B 0,C 180,E1 -15765.687,E2 -15765.687} C_VEL
LIN {X 0,Y 320.754,Z 272.203,A -85,B 0,C 180,E1 -15766.343,E2 -15766.343} C_VEL
LIN {X 0,Y 321.175,Z 258.817,A -85,B 0,C 180,E1 -15766.788,E2 -15766.788} C_VEL
LIN {X 0,Y 322.683,Z 185.061,A -85,B 0,C 180,E1 -15768.414,E2 -15768.414} C_VEL
LIN {X 0,Y 321.229,Z 178.58,A -85,B 0,C 180,E1 -15768.669,E2 -15768.669} C_VEL
LIN {X 0,Y 313.775,Z 158.923,A -85,B 0,C 180,E1 -15769.695,E2 -15769.695} C_VEL
LIN {X 0,Y 313.136,Z 157.063,A -85,B 0,C 180,E1 -15769.826,E2 -15769.826} C_VEL
LIN {X 0,Y 312.58,Z 154.55,A -85,B 0,C 180,E1 -15770.651,E2 -15770.651} C_VEL
LIN {X 0,Y 312.537,Z 154.555,A -85,B 0,C 180,E1 -15773.875,E2 -15773.875} C_VEL
LIN {X 0,Y 312.553,Z 154.551,A -85,B 0,C 180,E1 -15776.724,E2 -15776.724} C_VEL
LIN {X 0,Y 312.543,Z 154.552,A -85,B 0,C 180,E1 -15779.648,E2 -15779.648} C_VEL
LIN {X 0,Y 312.516,Z 154.555,A -85,B 0,C 180,E1 -15783.687,E2 -15783.687} C_VEL
LIN {X 0,Y 312.533,Z 154.552,A -85,B 0,C 180,E1 -15787.382,E2 -15787.382} C_VEL
LIN {X 0,Y 312.485,Z 154.557,A -85,B 0,C 180,E1 -15790.671,E2 -15790.671} C_VEL
LIN {X 0,Y 311.825,Z 154.643,A -85,B 0,C 180,E1 -15791.747,E2 -15791.747} C_VEL
LIN {X 0,Y 308.975,Z 154.998,A -85,B 0,C 180,E1 -15793.498,E2 -15793.498} C_VEL
